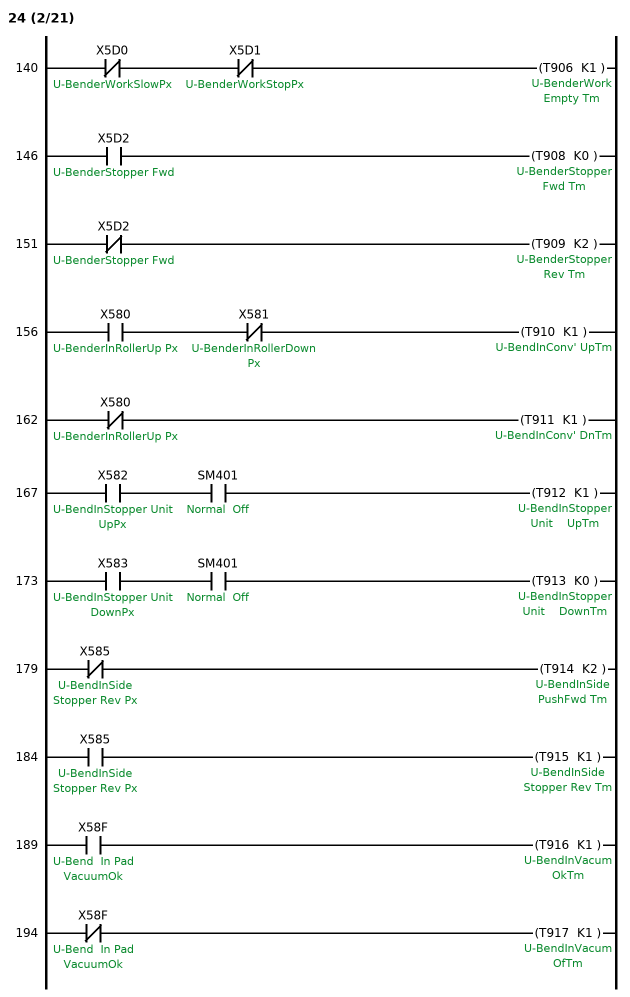
140   LDI     X5D0  ; U-BenderWorkSlowPx
      ANI     X5D1  ; U-BenderWorkStopPx
      OUT     T906 K1  ; U-BenderWork    Empty Tm
146   LD      X5D2  ; U-BenderStopper Fwd
      OUT     T908 K0  ; U-BenderStopper Fwd Tm
151   LDI     X5D2  ; U-BenderStopper Fwd
      OUT     T909 K2  ; U-BenderStopper Rev Tm
156   LD      X580  ; U-BenderInRollerUp Px
      ANI     X581  ; U-BenderInRollerDown Px
      OUT     T910 K1  ; U-BendInConv' UpTm
162   LDI     X580  ; U-BenderInRollerUp Px
      OUT     T911 K1  ; U-BendInConv' DnTm
167   LD      X582  ; U-BendInStopper Unit    UpPx
      AND     SM401  ; Normal  Off
      OUT     T912 K1  ; U-BendInStopper Unit    UpTm
173   LD      X583  ; U-BendInStopper Unit    DownPx
      AND     SM401  ; Normal  Off
      OUT     T913 K0  ; U-BendInStopper Unit    DownTm
179   LDI     X585  ; U-BendInSide    Stopper Rev Px
      OUT     T914 K2  ; U-BendInSide    PushFwd Tm
184   LD      X585  ; U-BendInSide    Stopper Rev Px
      OUT     T915 K1  ; U-BendInSide    Stopper Rev Tm
189   LD      X58F  ; U-Bend  In Pad  VacuumOk
      OUT     T916 K1  ; U-BendInVacum OkTm
194   LDI     X58F  ; U-Bend  In Pad  VacuumOk
      OUT     T917 K1  ; U-BendInVacum OfTm
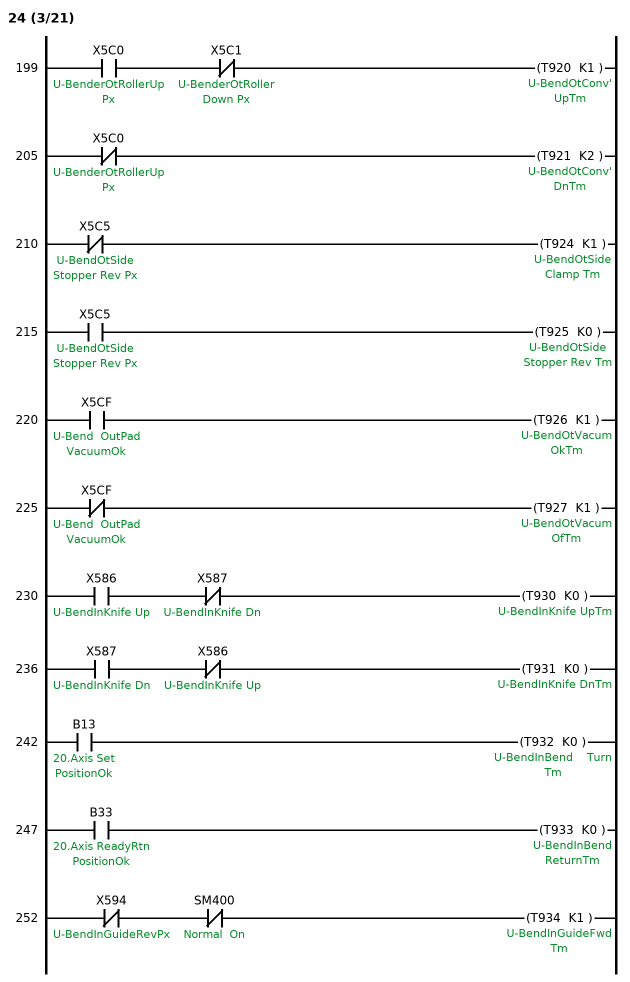
199   LD      X5C0  ; U-BenderOtRollerUp Px
      ANI     X5C1  ; U-BenderOtRollerDown Px
      OUT     T920 K1  ; U-BendOtConv' UpTm
205   LDI     X5C0  ; U-BenderOtRollerUp Px
      OUT     T921 K2  ; U-BendOtConv' DnTm
210   LDI     X5C5  ; U-BendOtSide    Stopper Rev Px
      OUT     T924 K1  ; U-BendOtSide    Clamp Tm
215   LD      X5C5  ; U-BendOtSide    Stopper Rev Px
      OUT     T925 K0  ; U-BendOtSide    Stopper Rev Tm
220   LD      X5CF  ; U-Bend  OutPad  VacuumOk
      OUT     T926 K1  ; U-BendOtVacum OkTm
225   LDI     X5CF  ; U-Bend  OutPad  VacuumOk
      OUT     T927 K1  ; U-BendOtVacum OfTm
230   LD      X586  ; U-BendInKnife Up
      ANI     X587  ; U-BendInKnife Dn
      OUT     T930 K0  ; U-BendInKnife UpTm
236   LD      X587  ; U-BendInKnife Dn
      ANI     X586  ; U-BendInKnife Up
      OUT     T931 K0  ; U-BendInKnife DnTm
242   LD      B13  ; 20.Axis Set     PositionOk
      OUT     T932 K0  ; U-BendInBend    Turn Tm
247   LD      B33  ; 20.Axis ReadyRtnPositionOk
      OUT     T933 K0  ; U-BendInBend    ReturnTm
252   LDI     X594  ; U-BendInGuideRevPx
      ANI     SM400  ; Normal  On
      OUT     T934 K1  ; U-BendInGuideFwdTm
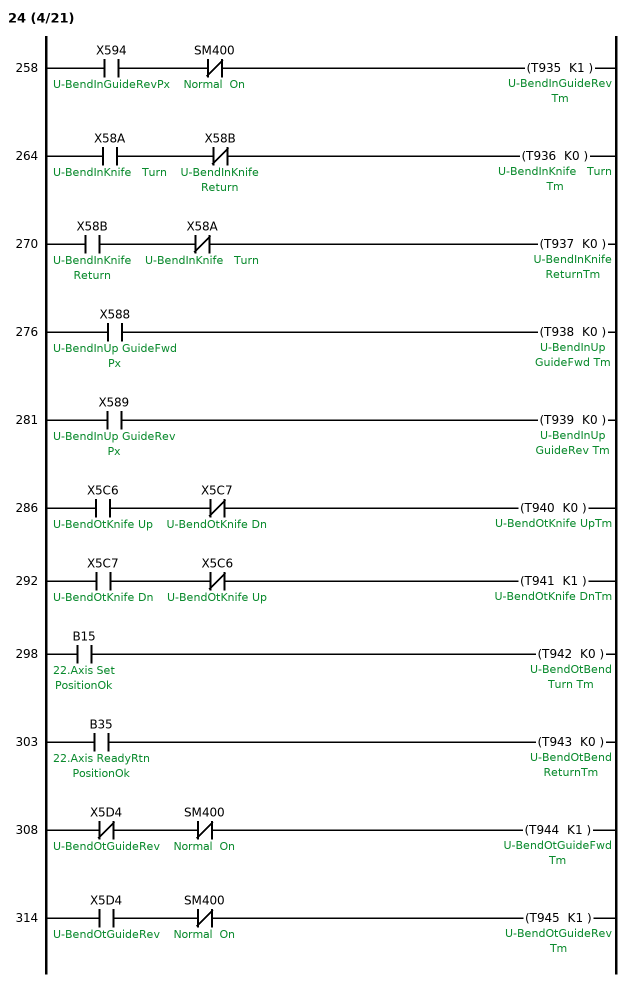
258   LD      X594  ; U-BendInGuideRevPx
      ANI     SM400  ; Normal  On
      OUT     T935 K1  ; U-BendInGuideRevTm
264   LD      X58A  ; U-BendInKnife   Turn
      ANI     X58B  ; U-BendInKnife   Return
      OUT     T936 K0  ; U-BendInKnife   Turn Tm
270   LD      X58B  ; U-BendInKnife   Return
      ANI     X58A  ; U-BendInKnife   Turn
      OUT     T937 K0  ; U-BendInKnife   ReturnTm
276   LD      X588  ; U-BendInUp GuideFwd Px
      OUT     T938 K0  ; U-BendInUp GuideFwd Tm
281   LD      X589  ; U-BendInUp GuideRev Px
      OUT     T939 K0  ; U-BendInUp GuideRev Tm
286   LD      X5C6  ; U-BendOtKnife Up
      ANI     X5C7  ; U-BendOtKnife Dn
      OUT     T940 K0  ; U-BendOtKnife UpTm
292   LD      X5C7  ; U-BendOtKnife Dn
      ANI     X5C6  ; U-BendOtKnife Up
      OUT     T941 K1  ; U-BendOtKnife DnTm
298   LD      B15  ; 22.Axis Set     PositionOk
      OUT     T942 K0  ; U-BendOtBend    Turn Tm
303   LD      B35  ; 22.Axis ReadyRtnPositionOk
      OUT     T943 K0  ; U-BendOtBend    ReturnTm
308   LDI     X5D4  ; U-BendOtGuideRev
      ANI     SM400  ; Normal  On
      OUT     T944 K1  ; U-BendOtGuideFwdTm
314   LD      X5D4  ; U-BendOtGuideRev
      ANI     SM400  ; Normal  On
      OUT     T945 K1  ; U-BendOtGuideRevTm
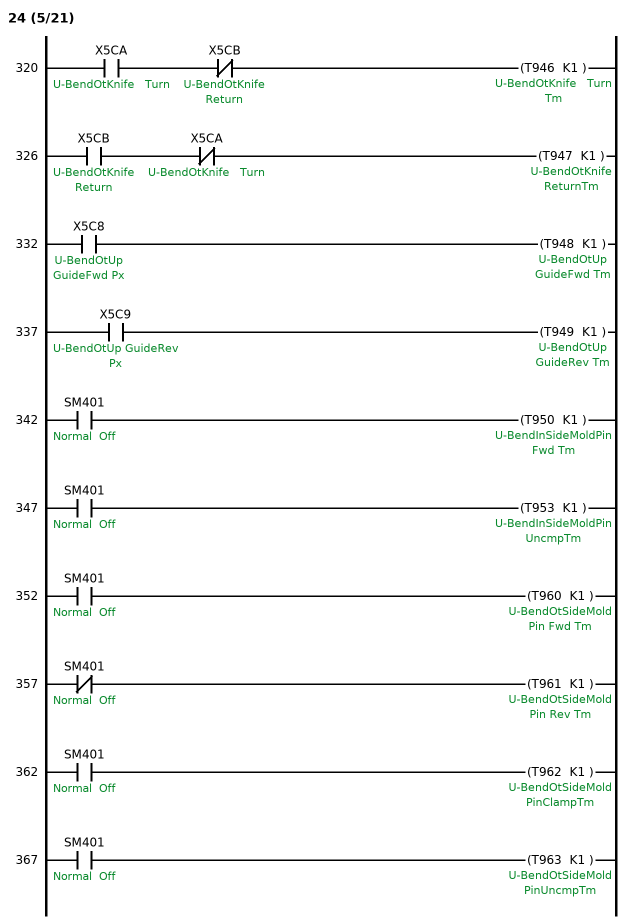
320   LD      X5CA  ; U-BendOtKnife   Turn
      ANI     X5CB  ; U-BendOtKnife   Return
      OUT     T946 K1  ; U-BendOtKnife   Turn Tm
326   LD      X5CB  ; U-BendOtKnife   Return
      ANI     X5CA  ; U-BendOtKnife   Turn
      OUT     T947 K1  ; U-BendOtKnife   ReturnTm
332   LD      X5C8  ; U-BendOtUp GuideFwd Px
      OUT     T948 K1  ; U-BendOtUp GuideFwd Tm
337   LD      X5C9  ; U-BendOtUp GuideRev Px
      OUT     T949 K1  ; U-BendOtUp GuideRev Tm
342   LD      SM401  ; Normal  Off
      OUT     T950 K1  ; U-BendInSideMoldPin Fwd Tm
347   LD      SM401  ; Normal  Off
      OUT     T953 K1  ; U-BendInSideMoldPinUncmpTm
352   LD      SM401  ; Normal  Off
      OUT     T960 K1  ; U-BendOtSideMoldPin Fwd Tm
357   LDI     SM401  ; Normal  Off
      OUT     T961 K1  ; U-BendOtSideMoldPin Rev Tm
362   LD      SM401  ; Normal  Off
      OUT     T962 K1  ; U-BendOtSideMoldPinClampTm
367   LD      SM401  ; Normal  Off
      OUT     T963 K1  ; U-BendOtSideMoldPinUncmpTm
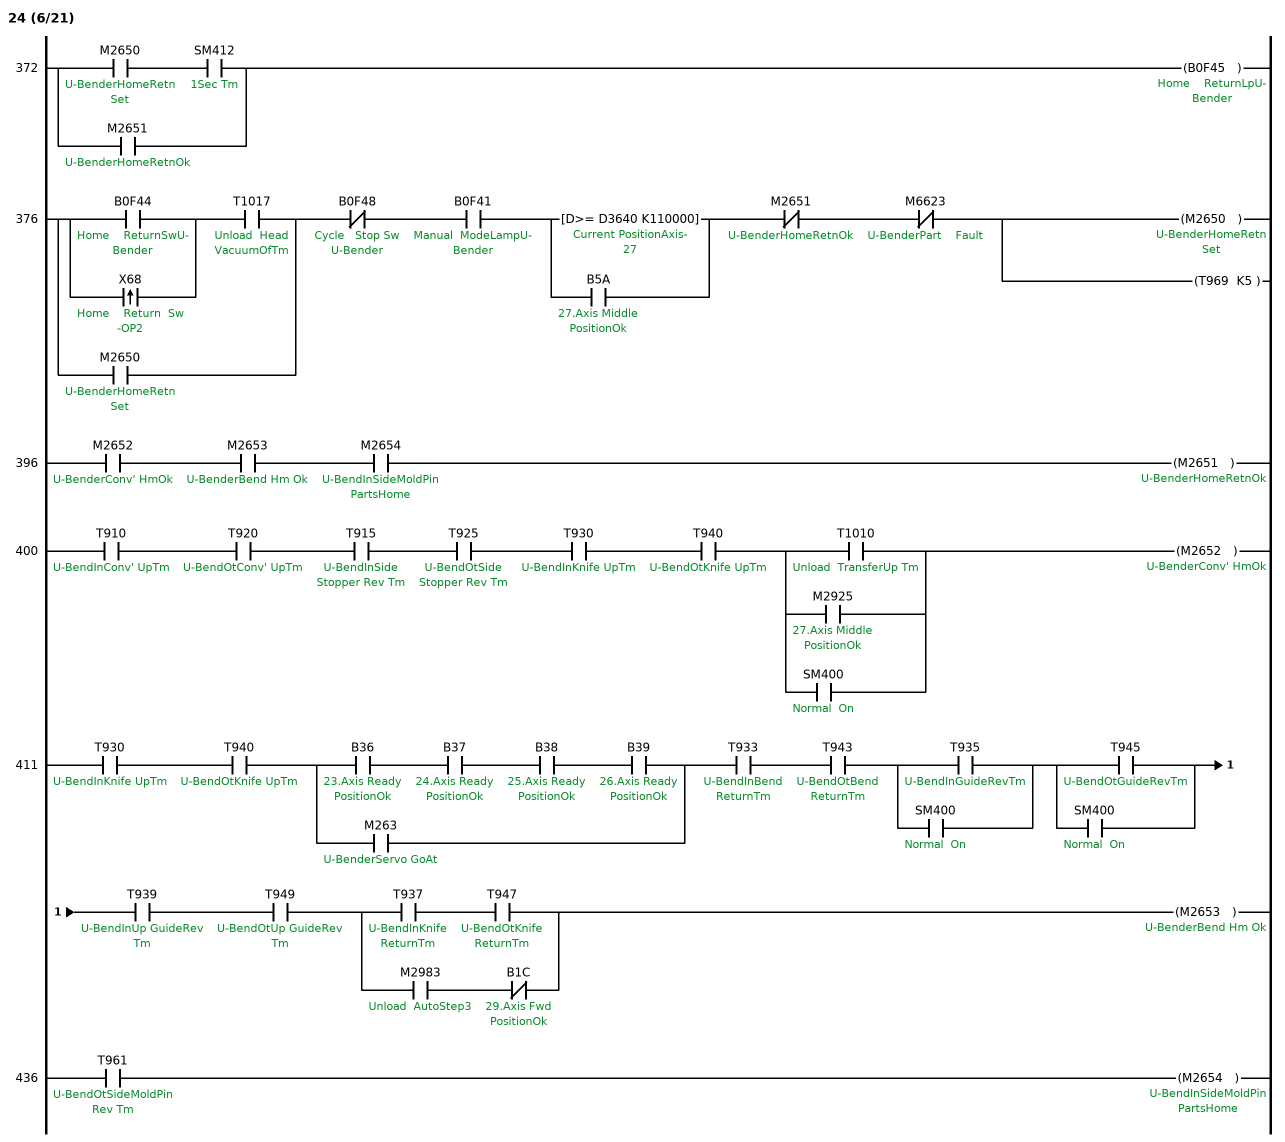
372   LD      M2650  ; U-BenderHomeRetnSet
      AND     SM412  ; 1Sec Tm
      OR      M2651  ; U-BenderHomeRetnOk
      OUT     B0F45  ; Home    ReturnLpU-Bender
376   LD      B0F44  ; Home    ReturnSwU-Bender
      ORP     X68  ; Home    Return  Sw -OP2
      AND     T1017  ; Unload  Head    VacuumOfTm
      OR      M2650  ; U-BenderHomeRetnSet
      ANI     B0F48  ; Cycle   Stop Sw U-Bender
      AND     B0F41  ; Manual  ModeLampU-Bender
      LDD>=   D3640 K110000  ; Current PositionAxis-27
      OR      B5A  ; 27.Axis Middle  PositionOk
      ANB
      ANI     M2651  ; U-BenderHomeRetnOk
      ANI     M6623  ; U-BenderPart    Fault
      OUT     M2650  ; U-BenderHomeRetnSet
      OUT     T969 K5
396   LD      M2652  ; U-BenderConv' HmOk
      AND     M2653  ; U-BenderBend Hm Ok
      AND     M2654  ; U-BendInSideMoldPinPartsHome
      OUT     M2651  ; U-BenderHomeRetnOk
400   LD      T910  ; U-BendInConv' UpTm
      AND     T920  ; U-BendOtConv' UpTm
      AND     T915  ; U-BendInSide    Stopper Rev Tm
      AND     T925  ; U-BendOtSide    Stopper Rev Tm
      AND     T930  ; U-BendInKnife UpTm
      AND     T940  ; U-BendOtKnife UpTm
      LD      T1010  ; Unload  TransferUp Tm
      OR      M2925  ; 27.Axis Middle  PositionOk
      OR      SM400  ; Normal  On
      ANB
      OUT     M2652  ; U-BenderConv' HmOk
411   LD      T930  ; U-BendInKnife UpTm
      AND     T940  ; U-BendOtKnife UpTm
      LD      B36  ; 23.Axis Ready   PositionOk
      AND     B37  ; 24.Axis Ready   PositionOk
      AND     B38  ; 25.Axis Ready   PositionOk
      AND     B39  ; 26.Axis Ready   PositionOk
      OR      M263  ; U-BenderServo GoAt
      ANB
      AND     T933  ; U-BendInBend    ReturnTm
      AND     T943  ; U-BendOtBend    ReturnTm
      LD      T935  ; U-BendInGuideRevTm
      OR      SM400  ; Normal  On
      ANB
      LD      T945  ; U-BendOtGuideRevTm
      OR      SM400  ; Normal  On
      ANB
      AND     T939  ; U-BendInUp GuideRev Tm
      AND     T949  ; U-BendOtUp GuideRev Tm
      LD      T937  ; U-BendInKnife   ReturnTm
      AND     T947  ; U-BendOtKnife   ReturnTm
      LD      M2983  ; Unload  AutoStep3
      ANI     B1C  ; 29.Axis Fwd     PositionOk
      ORB
      ANB
      OUT     M2653  ; U-BenderBend Hm Ok
436   LD      T961  ; U-BendOtSideMoldPin Rev Tm
      OUT     M2654  ; U-BendInSideMoldPinPartsHome
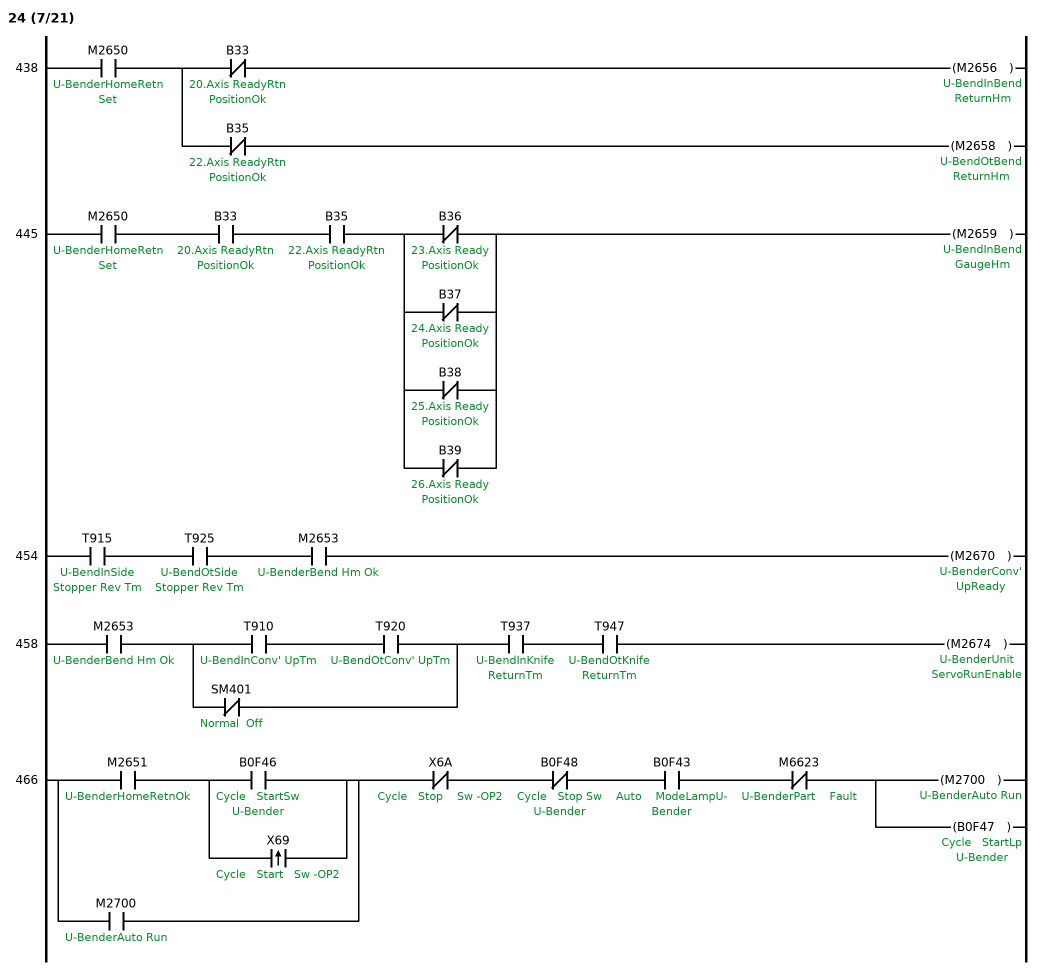
438   LD      M2650  ; U-BenderHomeRetnSet
      MPS
      ANI     B33  ; 20.Axis ReadyRtnPositionOk
      OUT     M2656  ; U-BendInBend    ReturnHm
      MPP
      ANI     B35  ; 22.Axis ReadyRtnPositionOk
      OUT     M2658  ; U-BendOtBend    ReturnHm
445   LD      M2650  ; U-BenderHomeRetnSet
      AND     B33  ; 20.Axis ReadyRtnPositionOk
      AND     B35  ; 22.Axis ReadyRtnPositionOk
      LDI     B36  ; 23.Axis Ready   PositionOk
      ORI     B37  ; 24.Axis Ready   PositionOk
      ORI     B38  ; 25.Axis Ready   PositionOk
      ORI     B39  ; 26.Axis Ready   PositionOk
      ANB
      OUT     M2659  ; U-BendInBend    GaugeHm
454   LD      T915  ; U-BendInSide    Stopper Rev Tm
      AND     T925  ; U-BendOtSide    Stopper Rev Tm
      AND     M2653  ; U-BenderBend Hm Ok
      OUT     M2670  ; U-BenderConv' UpReady
458   LD      M2653  ; U-BenderBend Hm Ok
      LD      T910  ; U-BendInConv' UpTm
      AND     T920  ; U-BendOtConv' UpTm
      ORI     SM401  ; Normal  Off
      ANB
      AND     T937  ; U-BendInKnife   ReturnTm
      AND     T947  ; U-BendOtKnife   ReturnTm
      OUT     M2674  ; U-BenderUnit    ServoRunEnable
466   LD      M2651  ; U-BenderHomeRetnOk
      LD      B0F46  ; Cycle   StartSw U-Bender
      ORP     X69  ; Cycle   Start   Sw -OP2
      ANB
      OR      M2700  ; U-BenderAuto Run
      ANI     X6A  ; Cycle   Stop    Sw -OP2
      ANI     B0F48  ; Cycle   Stop Sw U-Bender
      AND     B0F43  ; Auto    ModeLampU-Bender
      ANI     M6623  ; U-BenderPart    Fault
      OUT     M2700  ; U-BenderAuto Run
      OUT     B0F47  ; Cycle   StartLp U-Bender
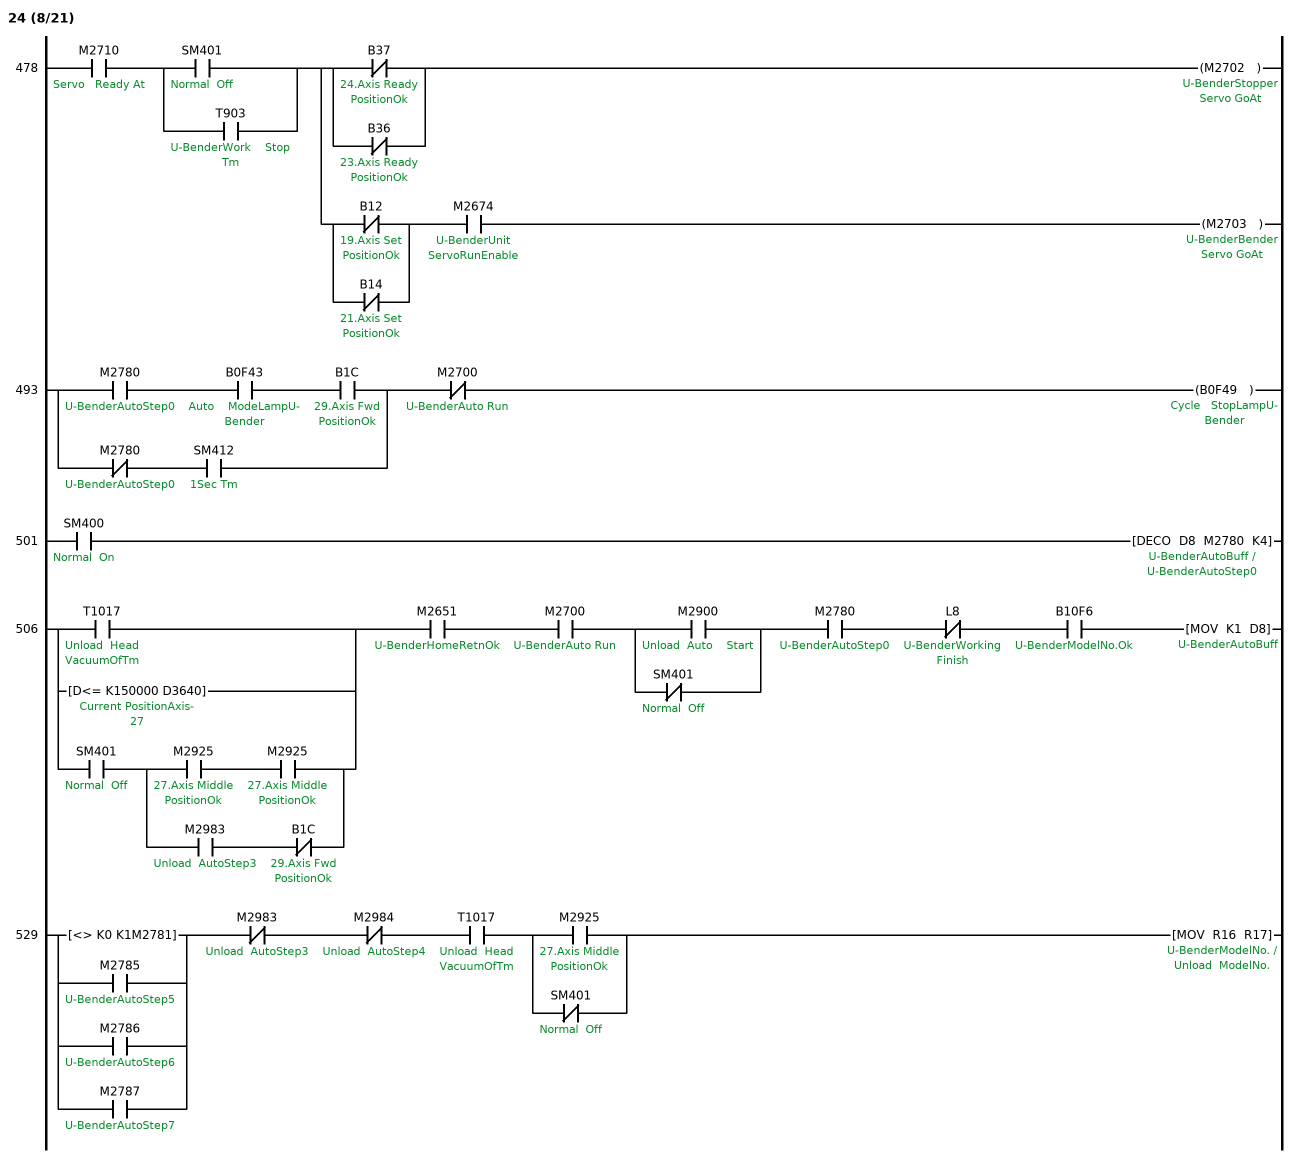
478   LD      M2710  ; Servo   Ready At
      LD      SM401  ; Normal  Off
      OR      T903  ; U-BenderWork    Stop Tm
      ANB
      MPS
      LDI     B37  ; 24.Axis Ready   PositionOk
      ORI     B36  ; 23.Axis Ready   PositionOk
      ANB
      OUT     M2702  ; U-BenderStopper Servo GoAt
      MPP
      LDI     B12  ; 19.Axis Set     PositionOk
      ORI     B14  ; 21.Axis Set     PositionOk
      ANB
      AND     M2674  ; U-BenderUnit    ServoRunEnable
      OUT     M2703  ; U-BenderBender  Servo GoAt
493   LD      M2780  ; U-BenderAutoStep0
      AND     B0F43  ; Auto    ModeLampU-Bender
      AND     B1C  ; 29.Axis Fwd     PositionOk
      LDI     M2780  ; U-BenderAutoStep0
      AND     SM412  ; 1Sec Tm
      ORB
      ANI     M2700  ; U-BenderAuto Run
      OUT     B0F49  ; Cycle   StopLampU-Bender
501   LD      SM400  ; Normal  On
      DECO    D8 M2780 K4  ; U-BenderAutoBuff
506   LD      T1017  ; Unload  Head    VacuumOfTm
      ORD<=   K150000 D3640  ; Current PositionAxis-27
      LD      SM401  ; Normal  Off
      LD      M2925  ; 27.Axis Middle  PositionOk
      AND     M2925  ; 27.Axis Middle  PositionOk
      LD      M2983  ; Unload  AutoStep3
      ANI     B1C  ; 29.Axis Fwd     PositionOk
      ORB
      ANB
      ORB
      AND     M2651  ; U-BenderHomeRetnOk
      AND     M2700  ; U-BenderAuto Run
      LD      M2900  ; Unload  Auto    Start
      ORI     SM401  ; Normal  Off
      ANB
      AND     M2780  ; U-BenderAutoStep0
      ANI     L8  ; U-BenderWorking Finish
      AND     B10F6  ; U-BenderModelNo.Ok
      MOV     K1 D8
529   LD<>    K0 K1M2781  ; U-BenderAutoStep1
      OR      M2785  ; U-BenderAutoStep5
      OR      M2786  ; U-BenderAutoStep6
      OR      M2787  ; U-BenderAutoStep7
      ANI     M2983  ; Unload  AutoStep3
      ANI     M2984  ; Unload  AutoStep4
      AND     T1017  ; Unload  Head    VacuumOfTm
      LD      M2925  ; 27.Axis Middle  PositionOk
      ORI     SM401  ; Normal  Off
      ANB
      MOV     R16 R17  ; U-BenderModelNo. / Unload  ModelNo.
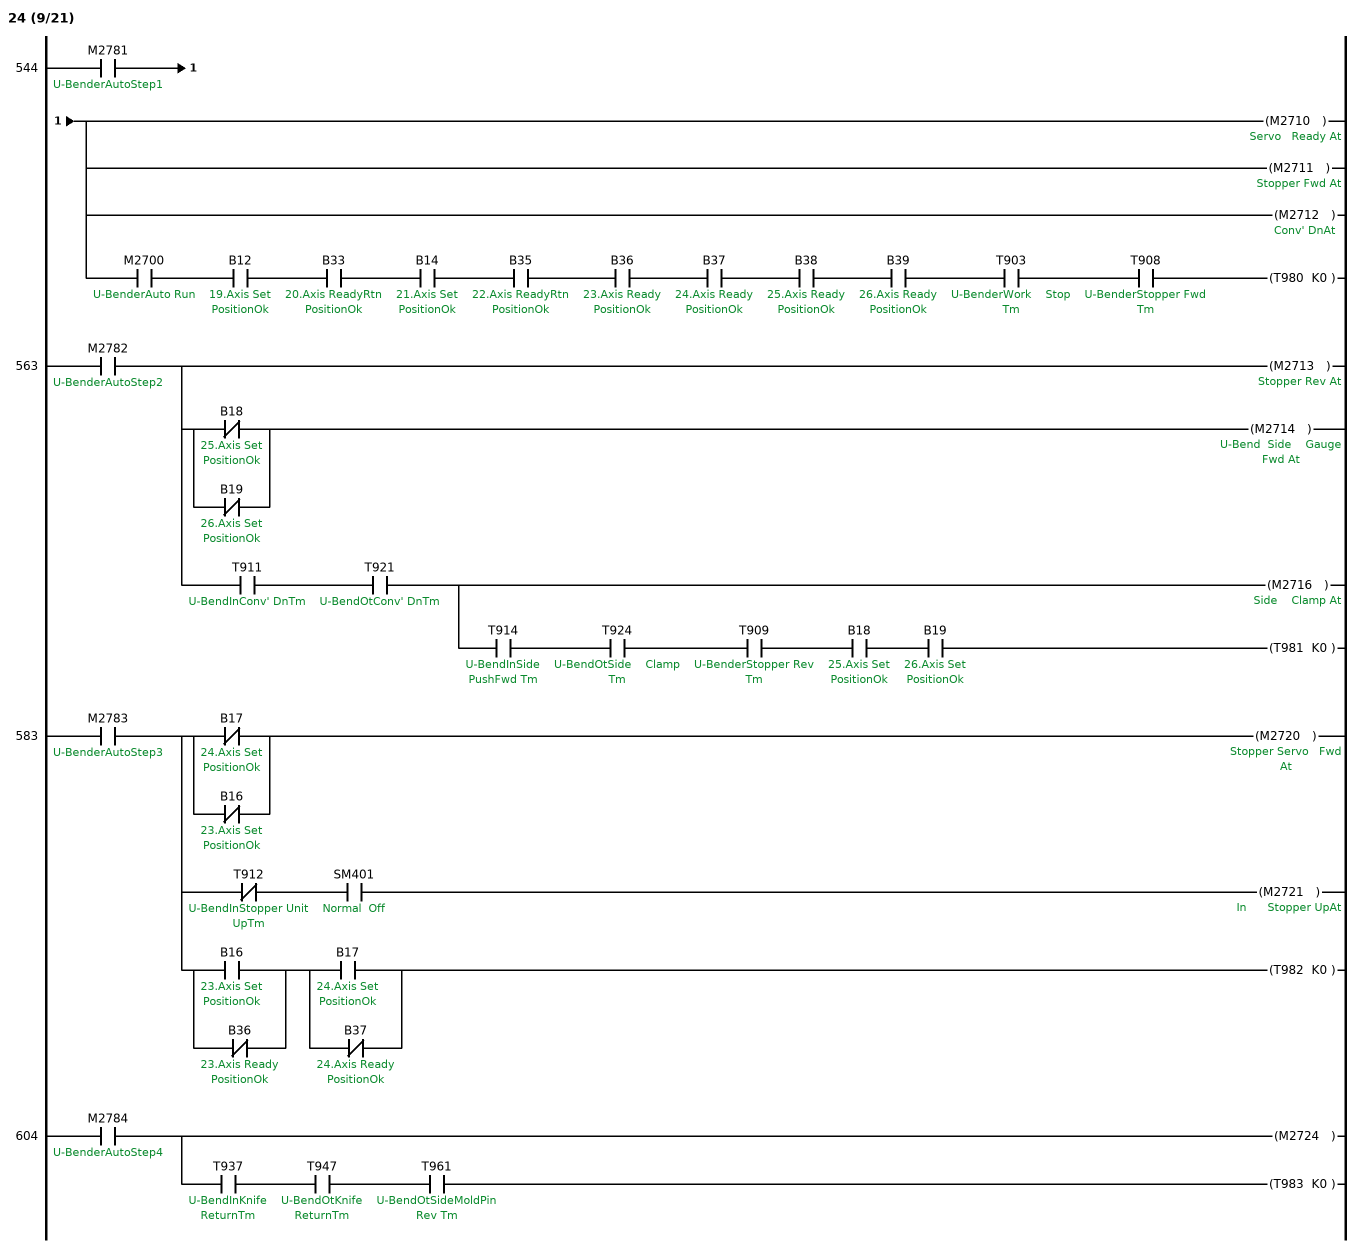
544   LD      M2781  ; U-BenderAutoStep1
      OUT     M2710  ; Servo   Ready At
      OUT     M2711  ; Stopper Fwd At
      OUT     M2712  ; Conv' DnAt
      AND     M2700  ; U-BenderAuto Run
      AND     B12  ; 19.Axis Set     PositionOk
      AND     B33  ; 20.Axis ReadyRtnPositionOk
      AND     B14  ; 21.Axis Set     PositionOk
      AND     B35  ; 22.Axis ReadyRtnPositionOk
      AND     B36  ; 23.Axis Ready   PositionOk
      AND     B37  ; 24.Axis Ready   PositionOk
      AND     B38  ; 25.Axis Ready   PositionOk
      AND     B39  ; 26.Axis Ready   PositionOk
      AND     T903  ; U-BenderWork    Stop Tm
      AND     T908  ; U-BenderStopper Fwd Tm
      OUT     T980 K0
563   LD      M2782  ; U-BenderAutoStep2
      OUT     M2713  ; Stopper Rev At
      MPS
      LDI     B18  ; 25.Axis Set     PositionOk
      ORI     B19  ; 26.Axis Set     PositionOk
      ANB
      OUT     M2714  ; U-Bend  Side    Gauge   Fwd At
      MPP
      AND     T911  ; U-BendInConv' DnTm
      AND     T921  ; U-BendOtConv' DnTm
      OUT     M2716  ; Side    Clamp At
      AND     T914  ; U-BendInSide    PushFwd Tm
      AND     T924  ; U-BendOtSide    Clamp Tm
      AND     T909  ; U-BenderStopper Rev Tm
      AND     B18  ; 25.Axis Set     PositionOk
      AND     B19  ; 26.Axis Set     PositionOk
      OUT     T981 K0
583   LD      M2783  ; U-BenderAutoStep3
      MPS
      LDI     B17  ; 24.Axis Set     PositionOk
      ORI     B16  ; 23.Axis Set     PositionOk
      ANB
      OUT     M2720  ; Stopper Servo   Fwd At
      MRD
      ANI     T912  ; U-BendInStopper Unit    UpTm
      AND     SM401  ; Normal  Off
      OUT     M2721  ; In      Stopper UpAt
      MPP
      LD      B16  ; 23.Axis Set     PositionOk
      ORI     B36  ; 23.Axis Ready   PositionOk
      ANB
      LD      B17  ; 24.Axis Set     PositionOk
      ORI     B37  ; 24.Axis Ready   PositionOk
      ANB
      OUT     T982 K0
604   LD      M2784  ; U-BenderAutoStep4
      OUT     M2724
      AND     T937  ; U-BendInKnife   ReturnTm
      AND     T947  ; U-BendOtKnife   ReturnTm
      AND     T961  ; U-BendOtSideMoldPin Rev Tm
      OUT     T983 K0
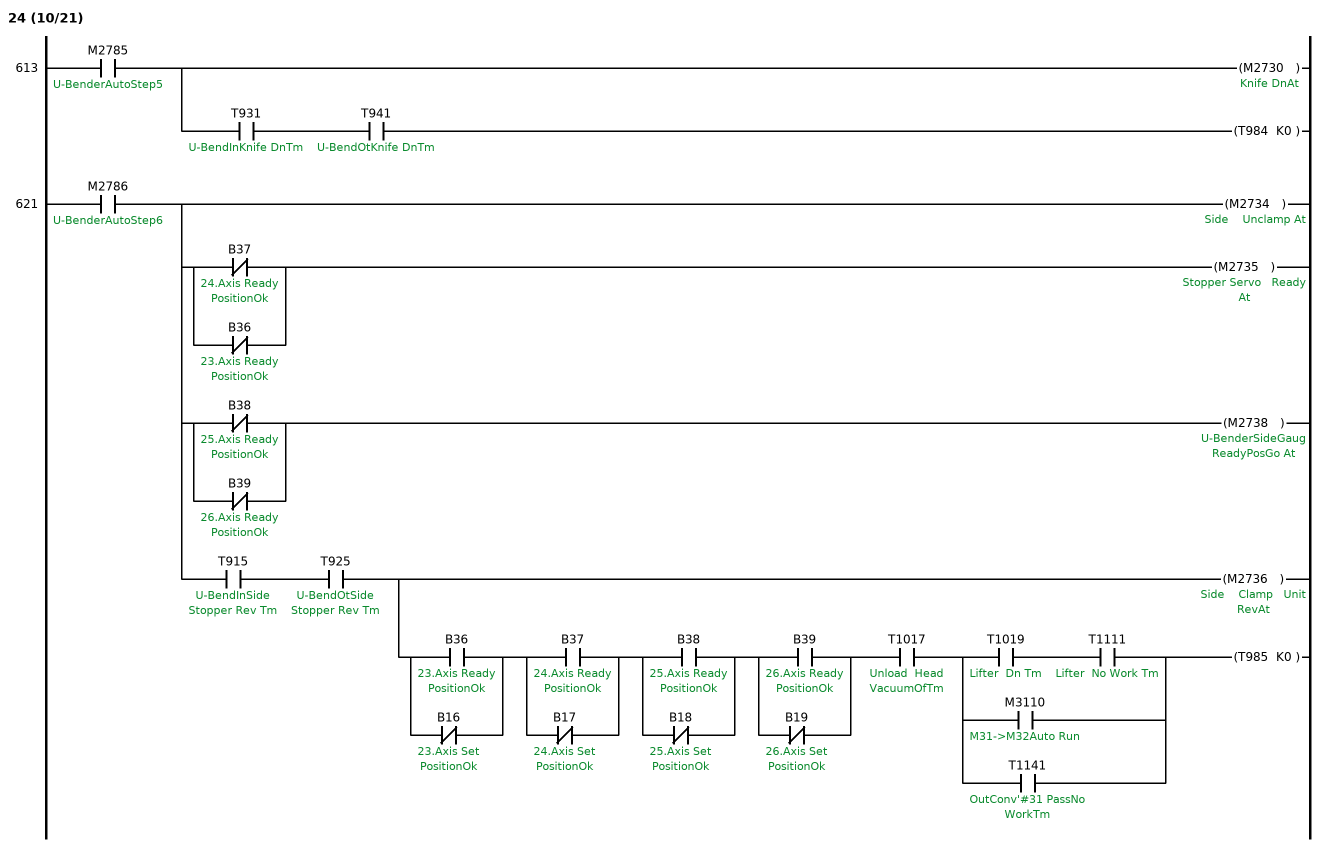
613   LD      M2785  ; U-BenderAutoStep5
      OUT     M2730  ; Knife DnAt
      AND     T931  ; U-BendInKnife DnTm
      AND     T941  ; U-BendOtKnife DnTm
      OUT     T984 K0
621   LD      M2786  ; U-BenderAutoStep6
      OUT     M2734  ; Side    Unclamp At
      MPS
      LDI     B37  ; 24.Axis Ready   PositionOk
      ORI     B36  ; 23.Axis Ready   PositionOk
      ANB
      OUT     M2735  ; Stopper Servo   Ready At
      MRD
      LDI     B38  ; 25.Axis Ready   PositionOk
      ORI     B39  ; 26.Axis Ready   PositionOk
      ANB
      OUT     M2738  ; U-BenderSideGaugReadyPosGo At
      MPP
      AND     T915  ; U-BendInSide    Stopper Rev Tm
      AND     T925  ; U-BendOtSide    Stopper Rev Tm
      OUT     M2736  ; Side    Clamp   Unit RevAt
      LD      B36  ; 23.Axis Ready   PositionOk
      ORI     B16  ; 23.Axis Set     PositionOk
      ANB
      LD      B37  ; 24.Axis Ready   PositionOk
      ORI     B17  ; 24.Axis Set     PositionOk
      ANB
      LD      B38  ; 25.Axis Ready   PositionOk
      ORI     B18  ; 25.Axis Set     PositionOk
      ANB
      LD      B39  ; 26.Axis Ready   PositionOk
      ORI     B19  ; 26.Axis Set     PositionOk
      ANB
      AND     T1017  ; Unload  Head    VacuumOfTm
      LD      T1019  ; Lifter  Dn Tm
      AND     T1111  ; Lifter  No Work Tm
      OR      M3110  ; M31->M32Auto Run
      OR      T1141  ; OutConv'#31 PassNo  WorkTm
      ANB
      OUT     T985 K0
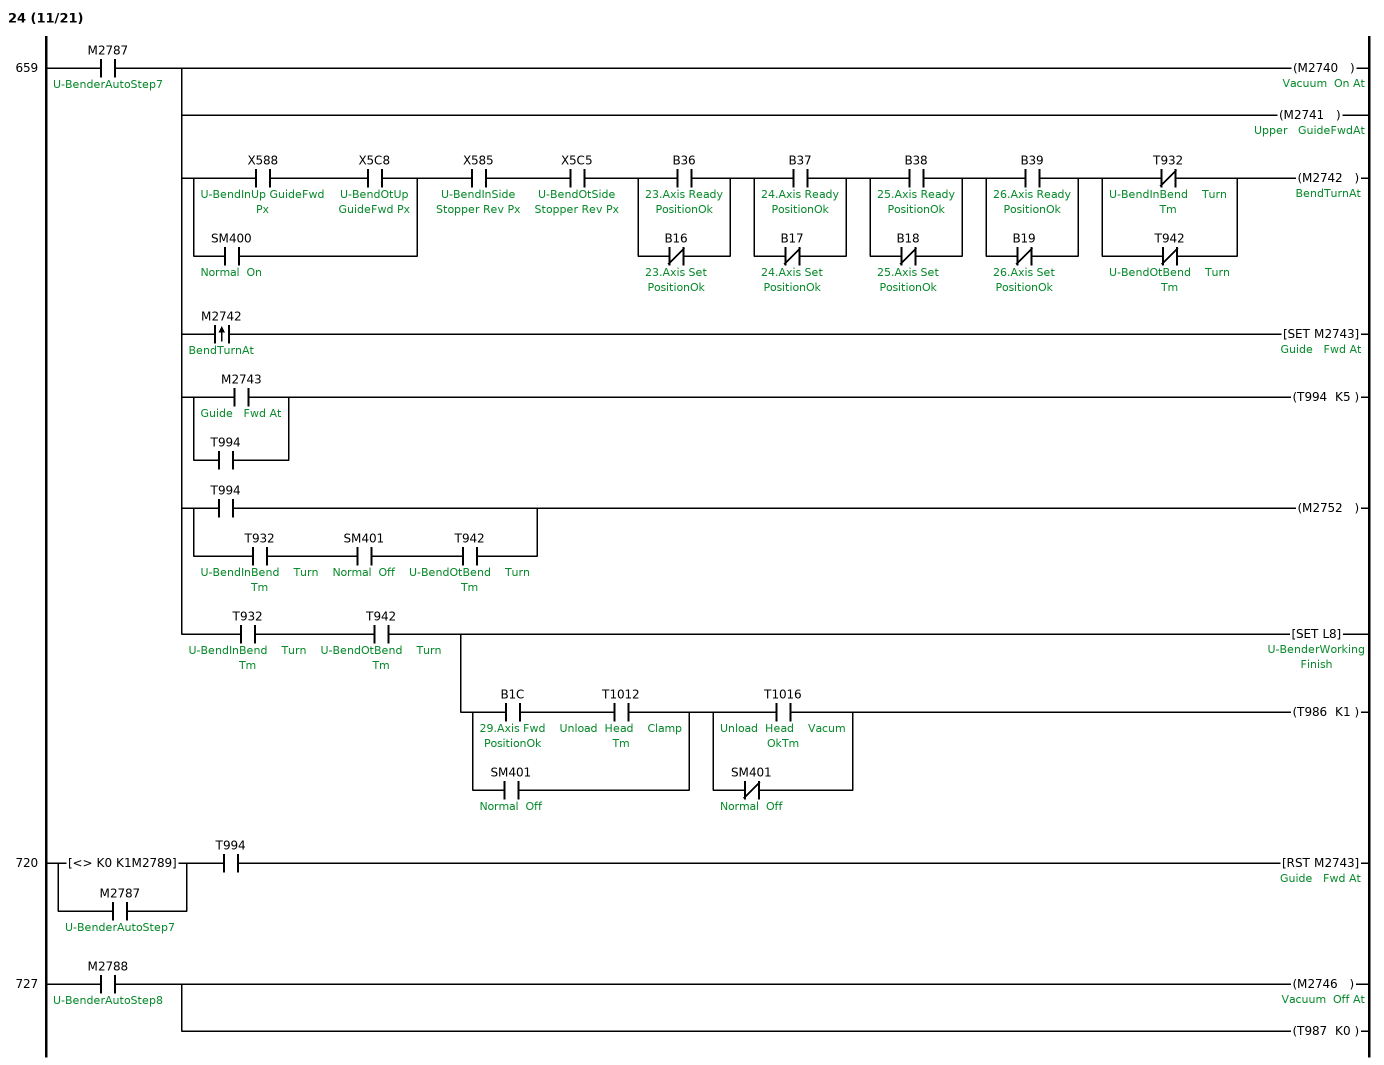
659   LD      M2787  ; U-BenderAutoStep7
      OUT     M2740  ; Vacuum  On At
      OUT     M2741  ; Upper   GuideFwdAt
      MPS
      LD      X588  ; U-BendInUp GuideFwd Px
      AND     X5C8  ; U-BendOtUp GuideFwd Px
      OR      SM400  ; Normal  On
      ANB
      AND     X585  ; U-BendInSide    Stopper Rev Px
      AND     X5C5  ; U-BendOtSide    Stopper Rev Px
      LD      B36  ; 23.Axis Ready   PositionOk
      ORI     B16  ; 23.Axis Set     PositionOk
      ANB
      LD      B37  ; 24.Axis Ready   PositionOk
      ORI     B17  ; 24.Axis Set     PositionOk
      ANB
      LD      B38  ; 25.Axis Ready   PositionOk
      ORI     B18  ; 25.Axis Set     PositionOk
      ANB
      LD      B39  ; 26.Axis Ready   PositionOk
      ORI     B19  ; 26.Axis Set     PositionOk
      ANB
      LDI     T932  ; U-BendInBend    Turn Tm
      ORI     T942  ; U-BendOtBend    Turn Tm
      ANB
      OUT     M2742  ; BendTurnAt
      MRD
      ANDP    M2742  ; BendTurnAt
      SET     M2743  ; Guide   Fwd At
      MRD
      LD      M2743  ; Guide   Fwd At
      OR      T994
      ANB
      OUT     T994 K5
      MRD
      LD      T994
      LD      T932  ; U-BendInBend    Turn Tm
      AND     SM401  ; Normal  Off
      AND     T942  ; U-BendOtBend    Turn Tm
      ORB
      ANB
      OUT     M2752
      MPP
      AND     T932  ; U-BendInBend    Turn Tm
      AND     T942  ; U-BendOtBend    Turn Tm
      SET     L8  ; U-BenderWorking Finish
      LD      B1C  ; 29.Axis Fwd     PositionOk
      AND     T1012  ; Unload  Head    Clamp Tm
      OR      SM401  ; Normal  Off
      ANB
      LD      T1016  ; Unload  Head    Vacum OkTm
      ORI     SM401  ; Normal  Off
      ANB
      OUT     T986 K1
720   LD<>    K0 K1M2789  ; U-BenderAutoStep9
      OR      M2787  ; U-BenderAutoStep7
      AND     T994
      RST     M2743  ; Guide   Fwd At
727   LD      M2788  ; U-BenderAutoStep8
      OUT     M2746  ; Vacuum  Off At
      OUT     T987 K0
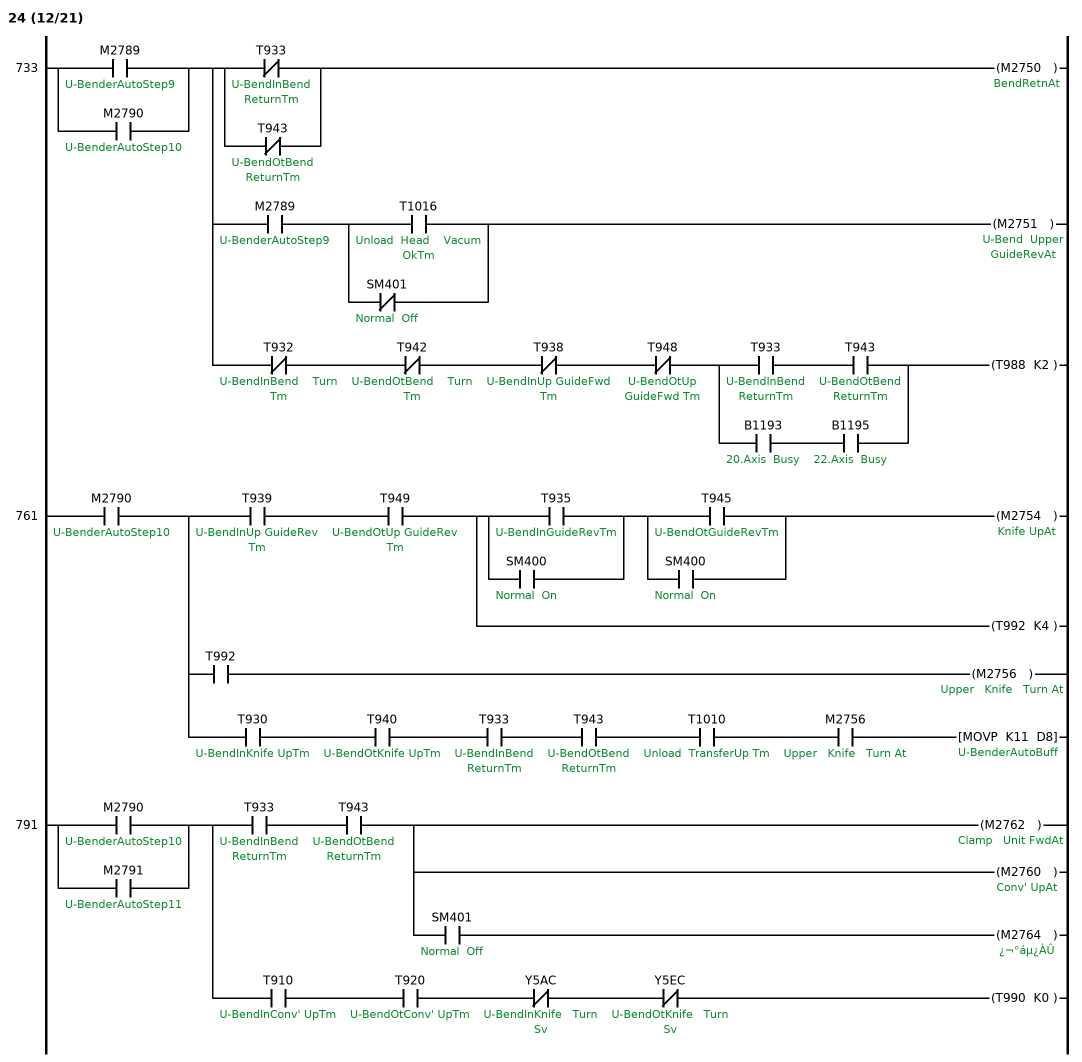
733   LD      M2789  ; U-BenderAutoStep9
      OR      M2790  ; U-BenderAutoStep10
      MPS
      LDI     T933  ; U-BendInBend    ReturnTm
      ORI     T943  ; U-BendOtBend    ReturnTm
      ANB
      OUT     M2750  ; BendRetnAt
      MRD
      AND     M2789  ; U-BenderAutoStep9
      LD      T1016  ; Unload  Head    Vacum OkTm
      ORI     SM401  ; Normal  Off
      ANB
      OUT     M2751  ; U-Bend  Upper   GuideRevAt
      MPP
      ANI     T932  ; U-BendInBend    Turn Tm
      ANI     T942  ; U-BendOtBend    Turn Tm
      ANI     T938  ; U-BendInUp GuideFwd Tm
      ANI     T948  ; U-BendOtUp GuideFwd Tm
      LD      T933  ; U-BendInBend    ReturnTm
      AND     T943  ; U-BendOtBend    ReturnTm
      LD      B1193  ; 20.Axis  Busy
      AND     B1195  ; 22.Axis  Busy
      ORB
      ANB
      OUT     T988 K2
761   LD      M2790  ; U-BenderAutoStep10
      MPS
      AND     T939  ; U-BendInUp GuideRev Tm
      AND     T949  ; U-BendOtUp GuideRev Tm
      MPS
      LD      T935  ; U-BendInGuideRevTm
      OR      SM400  ; Normal  On
      ANB
      LD      T945  ; U-BendOtGuideRevTm
      OR      SM400  ; Normal  On
      ANB
      OUT     M2754  ; Knife UpAt
      MPP
      OUT     T992 K4
      MRD
      AND     T992
      OUT     M2756  ; Upper   Knife   Turn At
      MPP
      AND     T930  ; U-BendInKnife UpTm
      AND     T940  ; U-BendOtKnife UpTm
      AND     T933  ; U-BendInBend    ReturnTm
      AND     T943  ; U-BendOtBend    ReturnTm
      AND     T1010  ; Unload  TransferUp Tm
      AND     M2756  ; Upper   Knife   Turn At
      MOVP    K11 D8
791   LD      M2790  ; U-BenderAutoStep10
      OR      M2791  ; U-BenderAutoStep11
      MPS
      AND     T933  ; U-BendInBend    ReturnTm
      AND     T943  ; U-BendOtBend    ReturnTm
      OUT     M2762  ; Clamp   Unit FwdAt
      OUT     M2760  ; Conv' UpAt
      AND     SM401  ; Normal  Off
      OUT     M2764  ; ¿¬°áµ¿ÀÛ
      MPP
      AND     T910  ; U-BendInConv' UpTm
      AND     T920  ; U-BendOtConv' UpTm
      ANI     Y5AC  ; U-BendInKnife   Turn Sv
      ANI     Y5EC  ; U-BendOtKnife   Turn Sv
      OUT     T990 K0
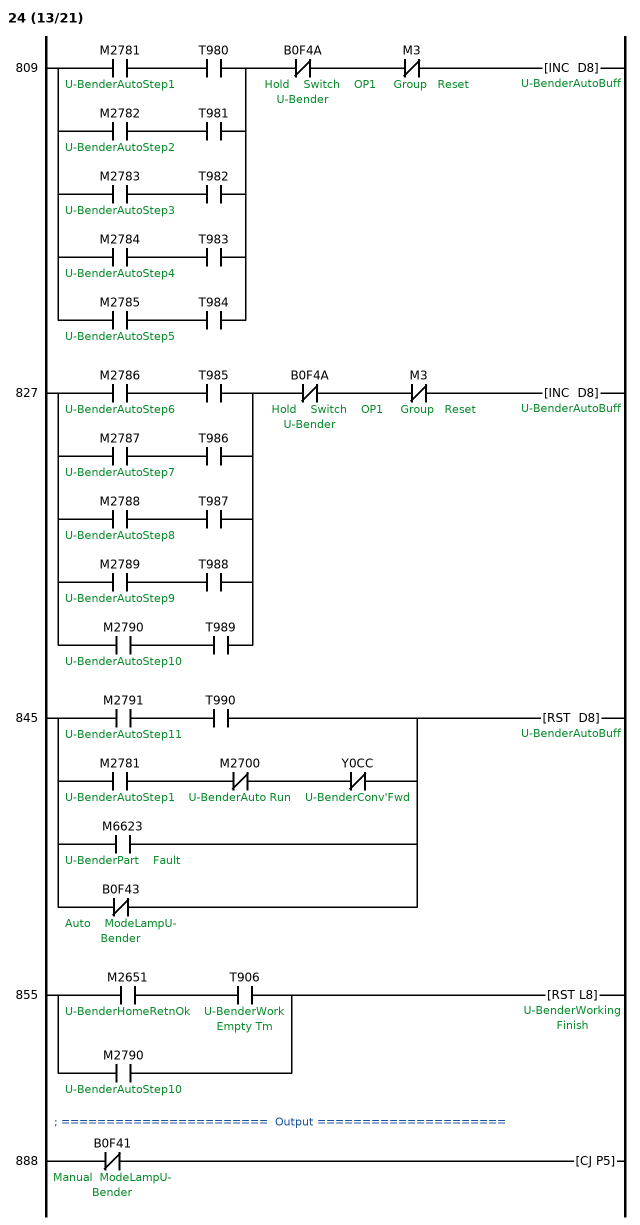
809   LD      M2781  ; U-BenderAutoStep1
      AND     T980
      LD      M2782  ; U-BenderAutoStep2
      AND     T981
      ORB
      LD      M2783  ; U-BenderAutoStep3
      AND     T982
      ORB
      LD      M2784  ; U-BenderAutoStep4
      AND     T983
      ORB
      LD      M2785  ; U-BenderAutoStep5
      AND     T984
      ORB
      ANI     B0F4A  ; Hold    Switch  U-Bender
      ANI     M3  ; OP1     Group   Reset
      INC     D8
827   LD      M2786  ; U-BenderAutoStep6
      AND     T985
      LD      M2787  ; U-BenderAutoStep7
      AND     T986
      ORB
      LD      M2788  ; U-BenderAutoStep8
      AND     T987
      ORB
      LD      M2789  ; U-BenderAutoStep9
      AND     T988
      ORB
      LD      M2790  ; U-BenderAutoStep10
      AND     T989
      ORB
      ANI     B0F4A  ; Hold    Switch  U-Bender
      ANI     M3  ; OP1     Group   Reset
      INC     D8
845   LD      M2791  ; U-BenderAutoStep11
      AND     T990
      LD      M2781  ; U-BenderAutoStep1
      ANI     M2700  ; U-BenderAuto Run
      ANI     Y0CC  ; U-BenderConv'Fwd
      ORB
      OR      M6623  ; U-BenderPart    Fault
      ORI     B0F43  ; Auto    ModeLampU-Bender
      RST     D8  ; U-BenderAutoBuff
855   LD      M2651  ; U-BenderHomeRetnOk
      AND     T906  ; U-BenderWork    Empty Tm
      OR      M2790  ; U-BenderAutoStep10
      RST     L8  ; U-BenderWorking Finish
; =======================  Output =====================
888   LDI     B0F41  ; Manual  ModeLampU-Bender
      CJ      P5
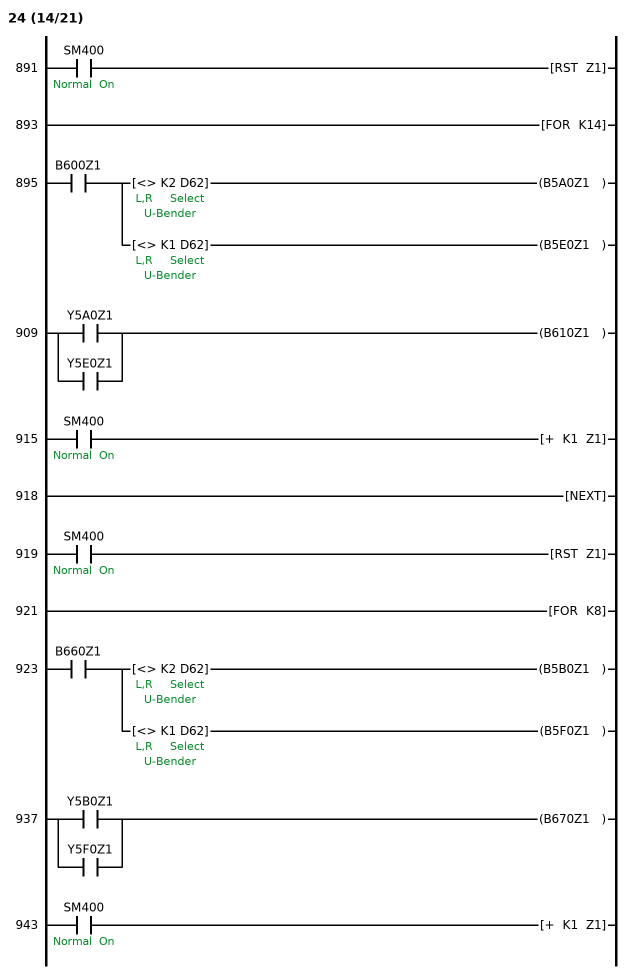
891   LD      SM400  ; Normal  On
      RST     Z1
893   FOR     K14
895   LD      B600Z1
      MPS
      AND<>   K2 D62  ; L,R     Select  U-Bender
      OUT     B5A0Z1
      MPP
      AND<>   K1 D62  ; L,R     Select  U-Bender
      OUT     B5E0Z1
909   LD      Y5A0Z1
      OR      Y5E0Z1
      OUT     B610Z1
915   LD      SM400  ; Normal  On
      +       K1 Z1
918   NEXT
919   LD      SM400  ; Normal  On
      RST     Z1
921   FOR     K8
923   LD      B660Z1
      MPS
      AND<>   K2 D62  ; L,R     Select  U-Bender
      OUT     B5B0Z1
      MPP
      AND<>   K1 D62  ; L,R     Select  U-Bender
      OUT     B5F0Z1
937   LD      Y5B0Z1
      OR      Y5F0Z1
      OUT     B670Z1
943   LD      SM400  ; Normal  On
      +       K1 Z1
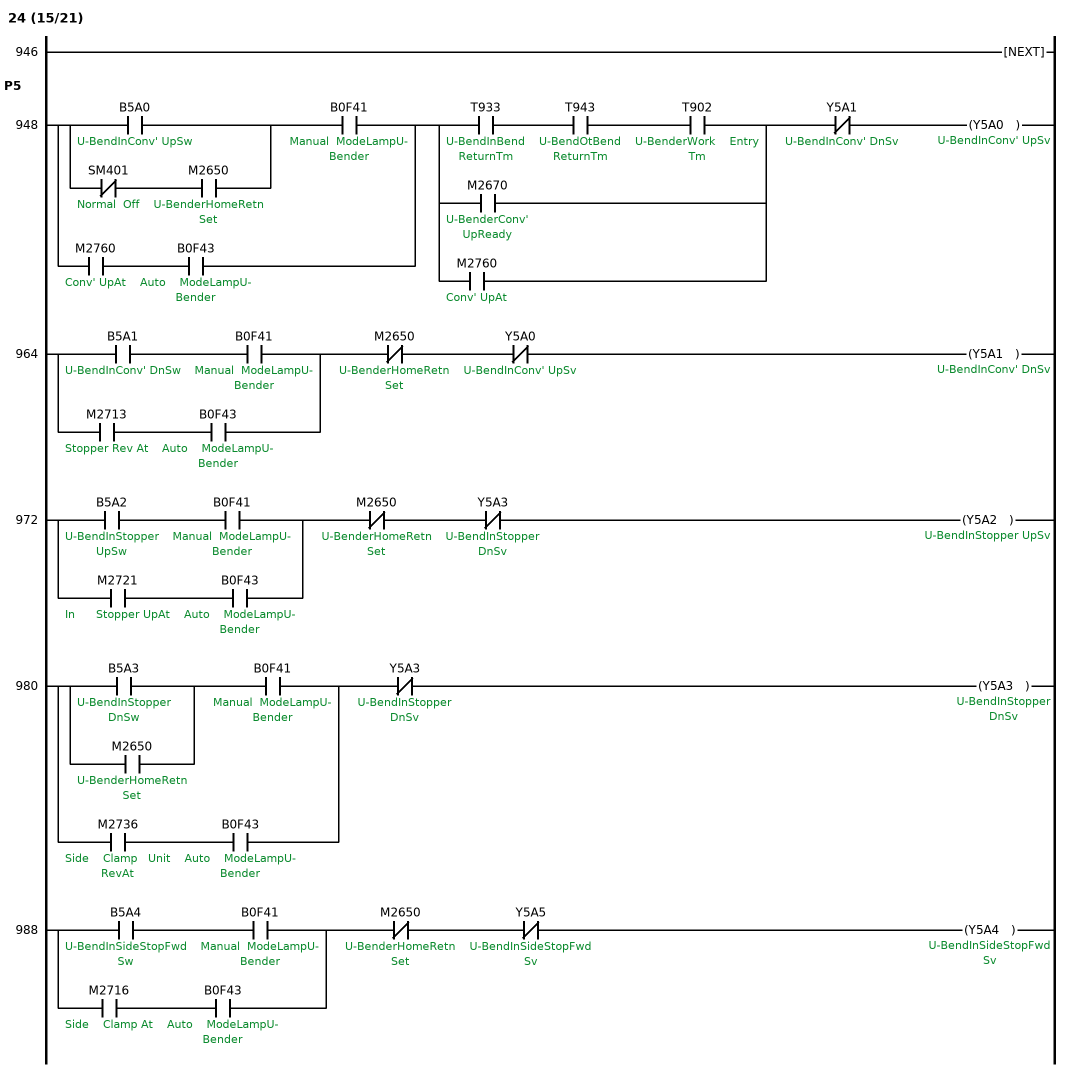
946   NEXT
      P5
948   LD      B5A0  ; U-BendInConv' UpSw
      LDI     SM401  ; Normal  Off
      AND     M2650  ; U-BenderHomeRetnSet
      ORB
      AND     B0F41  ; Manual  ModeLampU-Bender
      LD      M2760  ; Conv' UpAt
      AND     B0F43  ; Auto    ModeLampU-Bender
      ORB
      LD      T933  ; U-BendInBend    ReturnTm
      AND     T943  ; U-BendOtBend    ReturnTm
      AND     T902  ; U-BenderWork    Entry Tm
      OR      M2670  ; U-BenderConv' UpReady
      OR      M2760  ; Conv' UpAt
      ANB
      ANI     Y5A1  ; U-BendInConv' DnSv
      OUT     Y5A0  ; U-BendInConv' UpSv
964   LD      B5A1  ; U-BendInConv' DnSw
      AND     B0F41  ; Manual  ModeLampU-Bender
      LD      M2713  ; Stopper Rev At
      AND     B0F43  ; Auto    ModeLampU-Bender
      ORB
      ANI     M2650  ; U-BenderHomeRetnSet
      ANI     Y5A0  ; U-BendInConv' UpSv
      OUT     Y5A1  ; U-BendInConv' DnSv
972   LD      B5A2  ; U-BendInStopper UpSw
      AND     B0F41  ; Manual  ModeLampU-Bender
      LD      M2721  ; In      Stopper UpAt
      AND     B0F43  ; Auto    ModeLampU-Bender
      ORB
      ANI     M2650  ; U-BenderHomeRetnSet
      ANI     Y5A3  ; U-BendInStopper DnSv
      OUT     Y5A2  ; U-BendInStopper UpSv
980   LD      B5A3  ; U-BendInStopper DnSw
      OR      M2650  ; U-BenderHomeRetnSet
      AND     B0F41  ; Manual  ModeLampU-Bender
      LD      M2736  ; Side    Clamp   Unit RevAt
      AND     B0F43  ; Auto    ModeLampU-Bender
      ORB
      ANI     Y5A3  ; U-BendInStopper DnSv
      OUT     Y5A3  ; U-BendInStopper DnSv
988   LD      B5A4  ; U-BendInSideStopFwd     Sw
      AND     B0F41  ; Manual  ModeLampU-Bender
      LD      M2716  ; Side    Clamp At
      AND     B0F43  ; Auto    ModeLampU-Bender
      ORB
      ANI     M2650  ; U-BenderHomeRetnSet
      ANI     Y5A5  ; U-BendInSideStopFwd     Sv
      OUT     Y5A4  ; U-BendInSideStopFwd     Sv
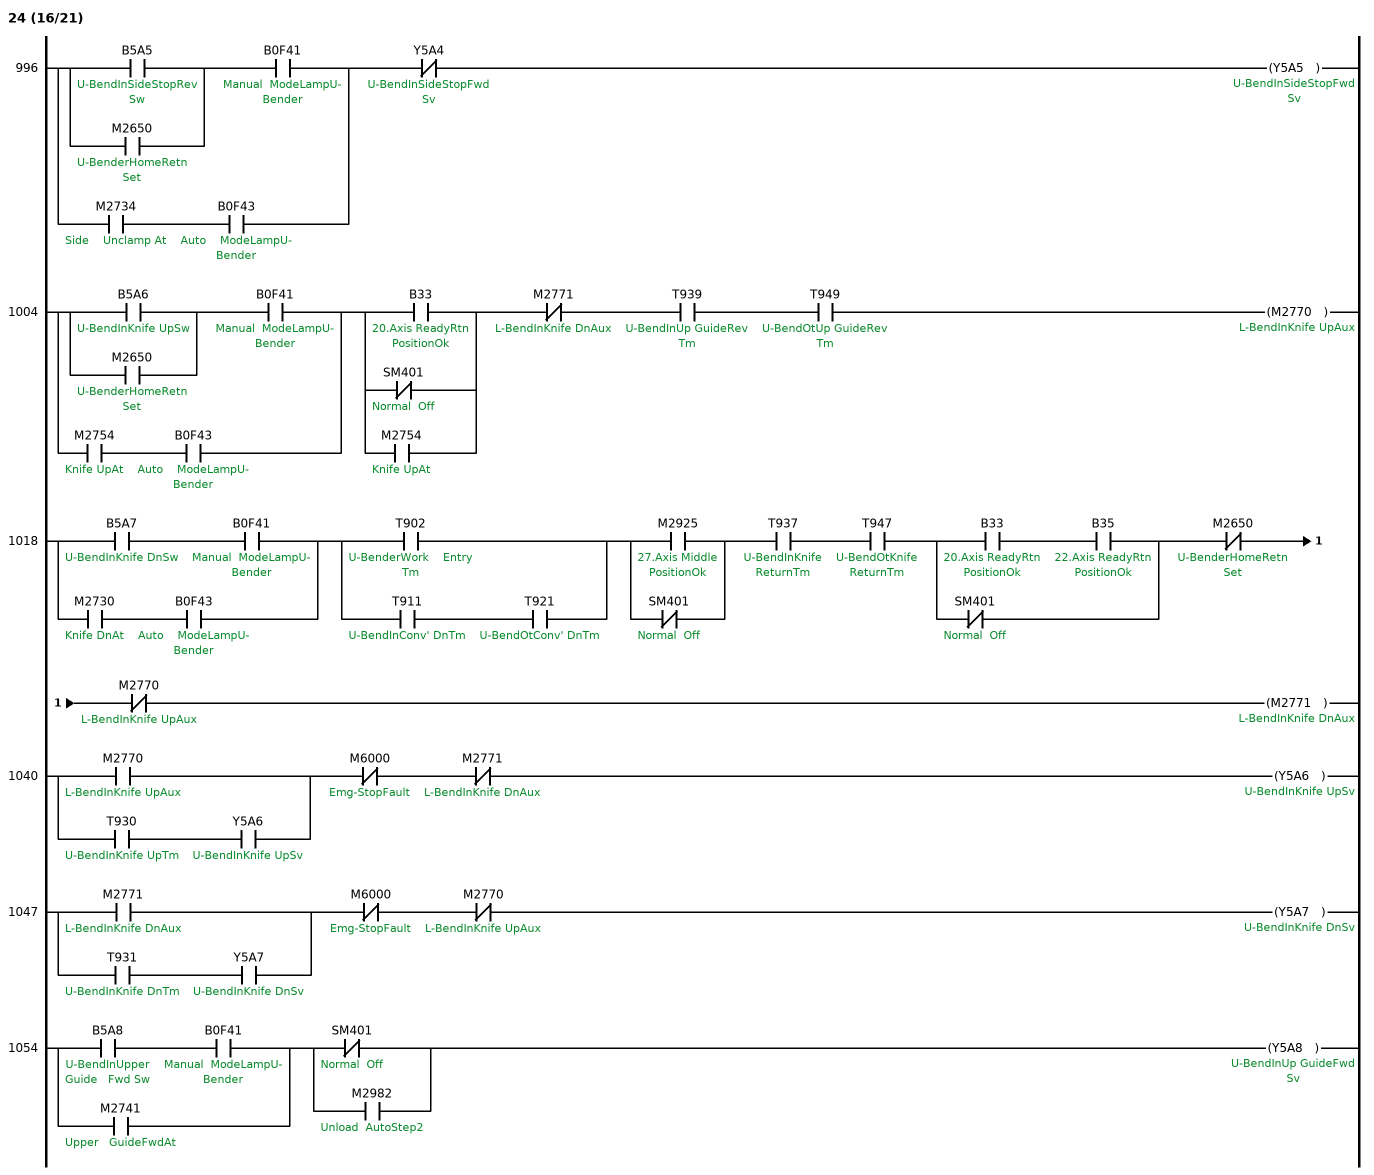
996   LD      B5A5  ; U-BendInSideStopRev     Sw
      OR      M2650  ; U-BenderHomeRetnSet
      AND     B0F41  ; Manual  ModeLampU-Bender
      LD      M2734  ; Side    Unclamp At
      AND     B0F43  ; Auto    ModeLampU-Bender
      ORB
      ANI     Y5A4  ; U-BendInSideStopFwd     Sv
      OUT     Y5A5  ; U-BendInSideStopFwd     Sv
1004  LD      B5A6  ; U-BendInKnife UpSw
      OR      M2650  ; U-BenderHomeRetnSet
      AND     B0F41  ; Manual  ModeLampU-Bender
      LD      M2754  ; Knife UpAt
      AND     B0F43  ; Auto    ModeLampU-Bender
      ORB
      LD      B33  ; 20.Axis ReadyRtnPositionOk
      ORI     SM401  ; Normal  Off
      OR      M2754  ; Knife UpAt
      ANB
      ANI     M2771  ; L-BendInKnife DnAux
      AND     T939  ; U-BendInUp GuideRev Tm
      AND     T949  ; U-BendOtUp GuideRev Tm
      OUT     M2770  ; L-BendInKnife UpAux
1018  LD      B5A7  ; U-BendInKnife DnSw
      AND     B0F41  ; Manual  ModeLampU-Bender
      LD      M2730  ; Knife DnAt
      AND     B0F43  ; Auto    ModeLampU-Bender
      ORB
      LD      T902  ; U-BenderWork    Entry Tm
      LD      T911  ; U-BendInConv' DnTm
      AND     T921  ; U-BendOtConv' DnTm
      ORB
      ANB
      LD      M2925  ; 27.Axis Middle  PositionOk
      ORI     SM401  ; Normal  Off
      ANB
      AND     T937  ; U-BendInKnife   ReturnTm
      AND     T947  ; U-BendOtKnife   ReturnTm
      LD      B33  ; 20.Axis ReadyRtnPositionOk
      AND     B35  ; 22.Axis ReadyRtnPositionOk
      ORI     SM401  ; Normal  Off
      ANB
      ANI     M2650  ; U-BenderHomeRetnSet
      ANI     M2770  ; L-BendInKnife UpAux
      OUT     M2771  ; L-BendInKnife DnAux
1040  LD      M2770  ; L-BendInKnife UpAux
      LD      T930  ; U-BendInKnife UpTm
      AND     Y5A6  ; U-BendInKnife UpSv
      ORB
      ANI     M6000  ; Emg-StopFault
      ANI     M2771  ; L-BendInKnife DnAux
      OUT     Y5A6  ; U-BendInKnife UpSv
1047  LD      M2771  ; L-BendInKnife DnAux
      LD      T931  ; U-BendInKnife DnTm
      AND     Y5A7  ; U-BendInKnife DnSv
      ORB
      ANI     M6000  ; Emg-StopFault
      ANI     M2770  ; L-BendInKnife UpAux
      OUT     Y5A7  ; U-BendInKnife DnSv
1054  LD      B5A8  ; U-BendInUpper   Guide   Fwd Sw
      AND     B0F41  ; Manual  ModeLampU-Bender
      OR      M2741  ; Upper   GuideFwdAt
      LDI     SM401  ; Normal  Off
      OR      M2982  ; Unload  AutoStep2
      ANB
      OUT     Y5A8  ; U-BendInUp GuideFwd Sv
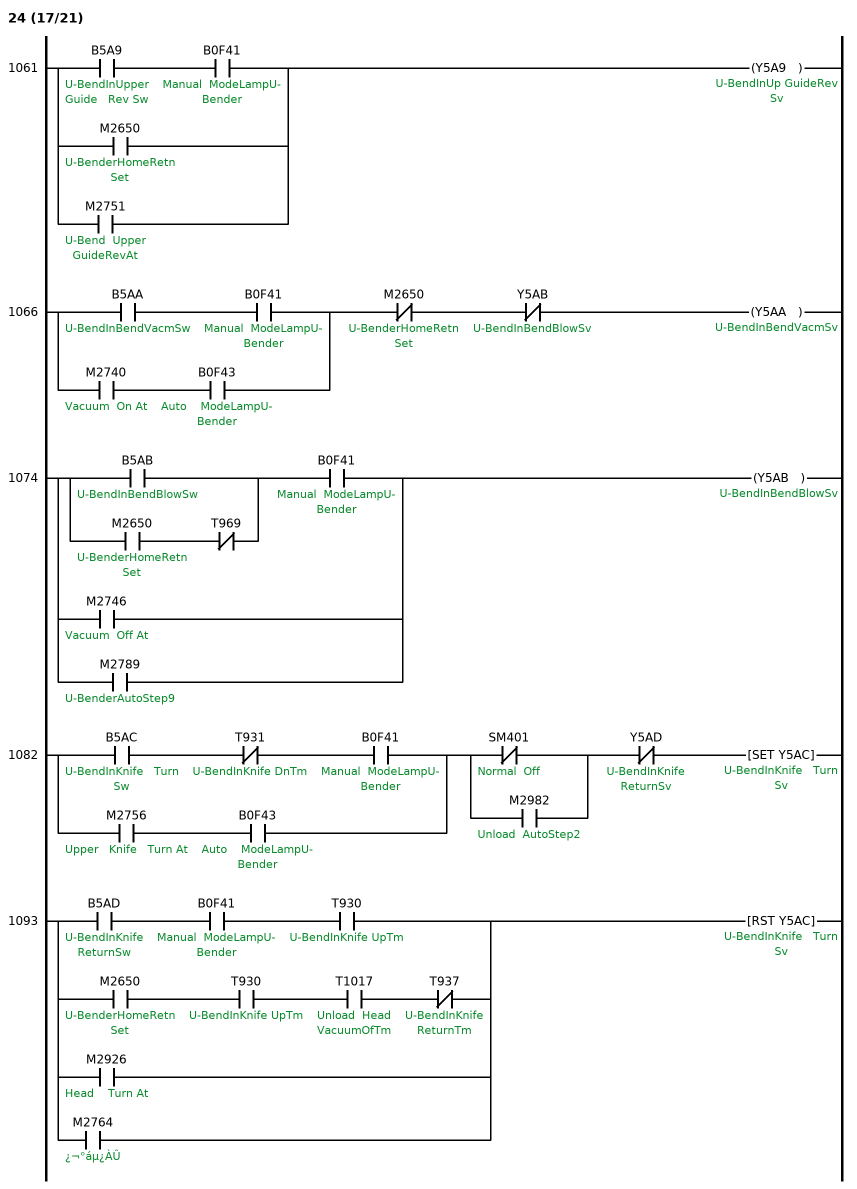
1061  LD      B5A9  ; U-BendInUpper   Guide   Rev Sw
      AND     B0F41  ; Manual  ModeLampU-Bender
      OR      M2650  ; U-BenderHomeRetnSet
      OR      M2751  ; U-Bend  Upper   GuideRevAt
      OUT     Y5A9  ; U-BendInUp GuideRev Sv
1066  LD      B5AA  ; U-BendInBendVacmSw
      AND     B0F41  ; Manual  ModeLampU-Bender
      LD      M2740  ; Vacuum  On At
      AND     B0F43  ; Auto    ModeLampU-Bender
      ORB
      ANI     M2650  ; U-BenderHomeRetnSet
      ANI     Y5AB  ; U-BendInBendBlowSv
      OUT     Y5AA  ; U-BendInBendVacmSv
1074  LD      B5AB  ; U-BendInBendBlowSw
      LD      M2650  ; U-BenderHomeRetnSet
      ANI     T969
      ORB
      AND     B0F41  ; Manual  ModeLampU-Bender
      OR      M2746  ; Vacuum  Off At
      OR      M2789  ; U-BenderAutoStep9
      OUT     Y5AB  ; U-BendInBendBlowSv
1082  LD      B5AC  ; U-BendInKnife   Turn Sw
      ANI     T931  ; U-BendInKnife DnTm
      AND     B0F41  ; Manual  ModeLampU-Bender
      LD      M2756  ; Upper   Knife   Turn At
      AND     B0F43  ; Auto    ModeLampU-Bender
      ORB
      LDI     SM401  ; Normal  Off
      OR      M2982  ; Unload  AutoStep2
      ANB
      ANI     Y5AD  ; U-BendInKnife   ReturnSv
      SET     Y5AC  ; U-BendInKnife   Turn Sv
1093  LD      B5AD  ; U-BendInKnife   ReturnSw
      AND     B0F41  ; Manual  ModeLampU-Bender
      AND     T930  ; U-BendInKnife UpTm
      LD      M2650  ; U-BenderHomeRetnSet
      AND     T930  ; U-BendInKnife UpTm
      AND     T1017  ; Unload  Head    VacuumOfTm
      ANI     T937  ; U-BendInKnife   ReturnTm
      ORB
      OR      M2926  ; Head    Turn At
      OR      M2764  ; ¿¬°áµ¿ÀÛ
      RST     Y5AC  ; U-BendInKnife   Turn Sv
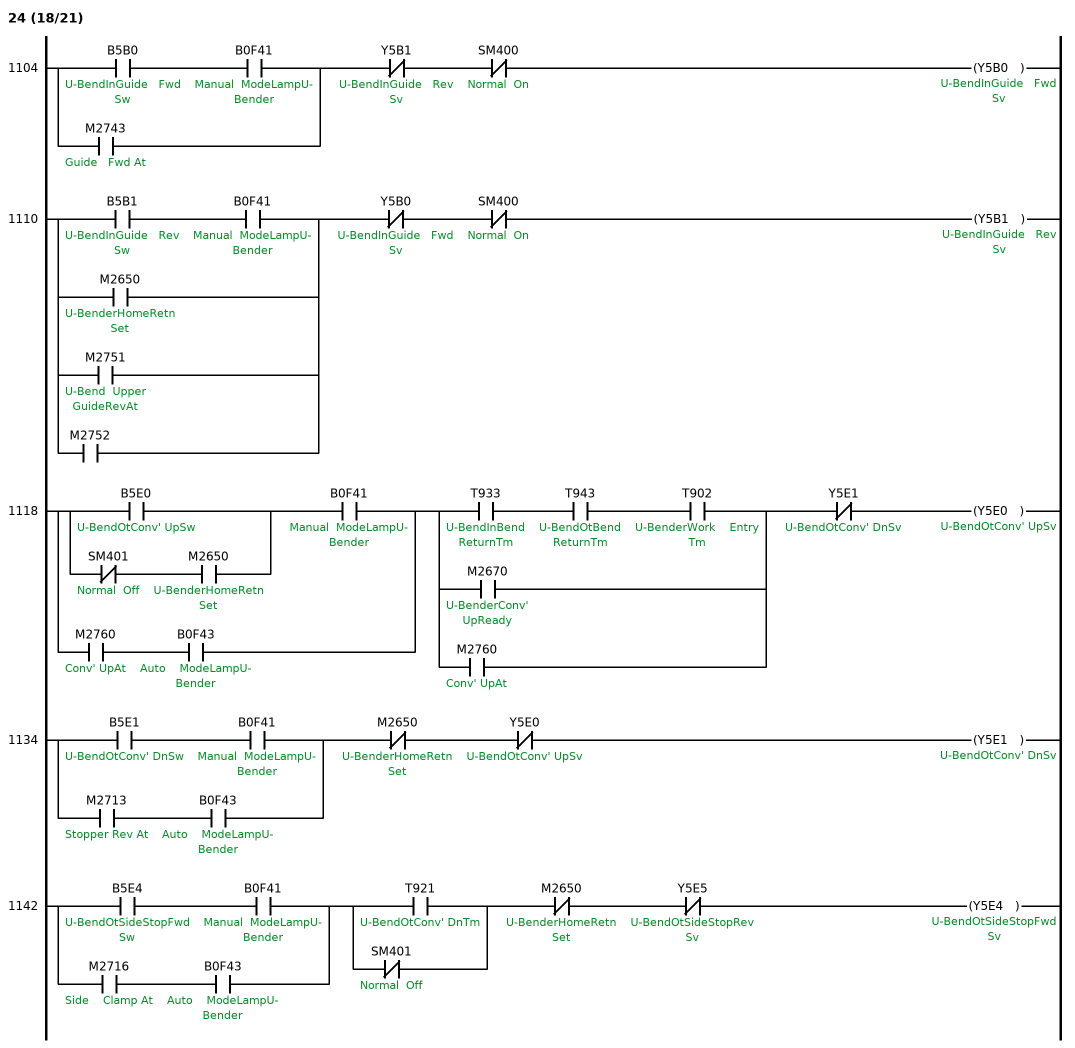
1104  LD      B5B0  ; U-BendInGuide   Fwd Sw
      AND     B0F41  ; Manual  ModeLampU-Bender
      OR      M2743  ; Guide   Fwd At
      ANI     Y5B1  ; U-BendInGuide   Rev Sv
      ANI     SM400  ; Normal  On
      OUT     Y5B0  ; U-BendInGuide   Fwd Sv
1110  LD      B5B1  ; U-BendInGuide   Rev Sw
      AND     B0F41  ; Manual  ModeLampU-Bender
      OR      M2650  ; U-BenderHomeRetnSet
      OR      M2751  ; U-Bend  Upper   GuideRevAt
      OR      M2752
      ANI     Y5B0  ; U-BendInGuide   Fwd Sv
      ANI     SM400  ; Normal  On
      OUT     Y5B1  ; U-BendInGuide   Rev Sv
1118  LD      B5E0  ; U-BendOtConv' UpSw
      LDI     SM401  ; Normal  Off
      AND     M2650  ; U-BenderHomeRetnSet
      ORB
      AND     B0F41  ; Manual  ModeLampU-Bender
      LD      M2760  ; Conv' UpAt
      AND     B0F43  ; Auto    ModeLampU-Bender
      ORB
      LD      T933  ; U-BendInBend    ReturnTm
      AND     T943  ; U-BendOtBend    ReturnTm
      AND     T902  ; U-BenderWork    Entry Tm
      OR      M2670  ; U-BenderConv' UpReady
      OR      M2760  ; Conv' UpAt
      ANB
      ANI     Y5E1  ; U-BendOtConv' DnSv
      OUT     Y5E0  ; U-BendOtConv' UpSv
1134  LD      B5E1  ; U-BendOtConv' DnSw
      AND     B0F41  ; Manual  ModeLampU-Bender
      LD      M2713  ; Stopper Rev At
      AND     B0F43  ; Auto    ModeLampU-Bender
      ORB
      ANI     M2650  ; U-BenderHomeRetnSet
      ANI     Y5E0  ; U-BendOtConv' UpSv
      OUT     Y5E1  ; U-BendOtConv' DnSv
1142  LD      B5E4  ; U-BendOtSideStopFwd     Sw
      AND     B0F41  ; Manual  ModeLampU-Bender
      LD      M2716  ; Side    Clamp At
      AND     B0F43  ; Auto    ModeLampU-Bender
      ORB
      LD      T921  ; U-BendOtConv' DnTm
      ORI     SM401  ; Normal  Off
      ANB
      ANI     M2650  ; U-BenderHomeRetnSet
      ANI     Y5E5  ; U-BendOtSideStopRev     Sv
      OUT     Y5E4  ; U-BendOtSideStopFwd     Sv
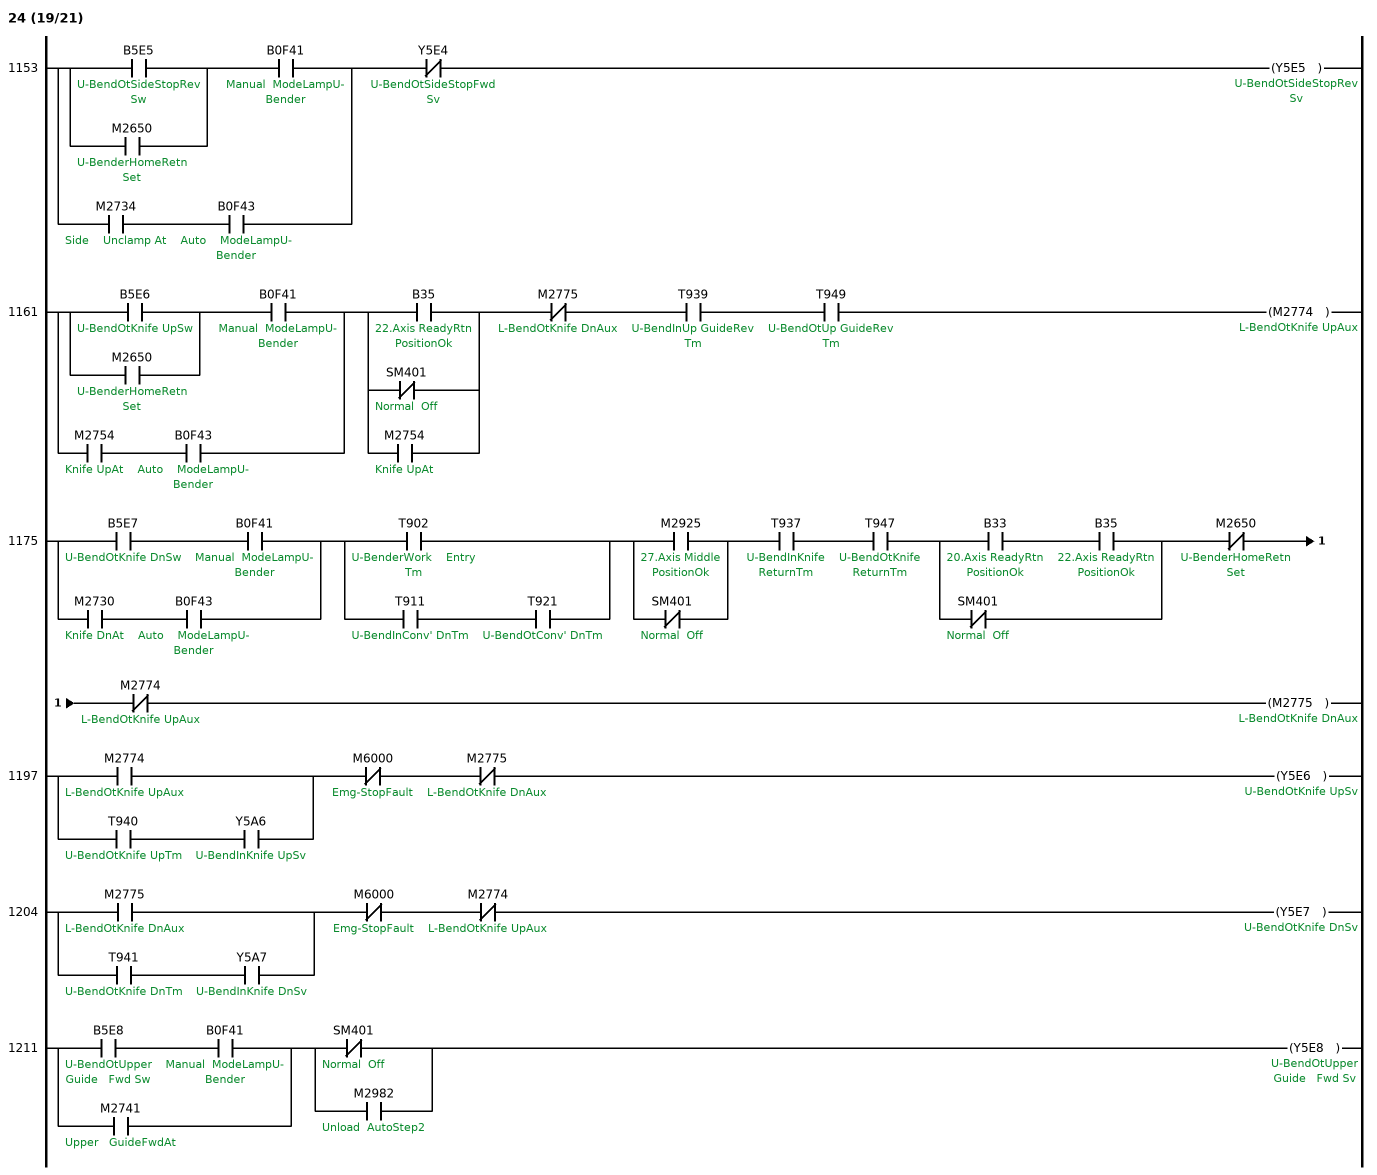
1153  LD      B5E5  ; U-BendOtSideStopRev     Sw
      OR      M2650  ; U-BenderHomeRetnSet
      AND     B0F41  ; Manual  ModeLampU-Bender
      LD      M2734  ; Side    Unclamp At
      AND     B0F43  ; Auto    ModeLampU-Bender
      ORB
      ANI     Y5E4  ; U-BendOtSideStopFwd     Sv
      OUT     Y5E5  ; U-BendOtSideStopRev     Sv
1161  LD      B5E6  ; U-BendOtKnife UpSw
      OR      M2650  ; U-BenderHomeRetnSet
      AND     B0F41  ; Manual  ModeLampU-Bender
      LD      M2754  ; Knife UpAt
      AND     B0F43  ; Auto    ModeLampU-Bender
      ORB
      LD      B35  ; 22.Axis ReadyRtnPositionOk
      ORI     SM401  ; Normal  Off
      OR      M2754  ; Knife UpAt
      ANB
      ANI     M2775  ; L-BendOtKnife DnAux
      AND     T939  ; U-BendInUp GuideRev Tm
      AND     T949  ; U-BendOtUp GuideRev Tm
      OUT     M2774  ; L-BendOtKnife UpAux
1175  LD      B5E7  ; U-BendOtKnife DnSw
      AND     B0F41  ; Manual  ModeLampU-Bender
      LD      M2730  ; Knife DnAt
      AND     B0F43  ; Auto    ModeLampU-Bender
      ORB
      LD      T902  ; U-BenderWork    Entry Tm
      LD      T911  ; U-BendInConv' DnTm
      AND     T921  ; U-BendOtConv' DnTm
      ORB
      ANB
      LD      M2925  ; 27.Axis Middle  PositionOk
      ORI     SM401  ; Normal  Off
      ANB
      AND     T937  ; U-BendInKnife   ReturnTm
      AND     T947  ; U-BendOtKnife   ReturnTm
      LD      B33  ; 20.Axis ReadyRtnPositionOk
      AND     B35  ; 22.Axis ReadyRtnPositionOk
      ORI     SM401  ; Normal  Off
      ANB
      ANI     M2650  ; U-BenderHomeRetnSet
      ANI     M2774  ; L-BendOtKnife UpAux
      OUT     M2775  ; L-BendOtKnife DnAux
1197  LD      M2774  ; L-BendOtKnife UpAux
      LD      T940  ; U-BendOtKnife UpTm
      AND     Y5A6  ; U-BendInKnife UpSv
      ORB
      ANI     M6000  ; Emg-StopFault
      ANI     M2775  ; L-BendOtKnife DnAux
      OUT     Y5E6  ; U-BendOtKnife UpSv
1204  LD      M2775  ; L-BendOtKnife DnAux
      LD      T941  ; U-BendOtKnife DnTm
      AND     Y5A7  ; U-BendInKnife DnSv
      ORB
      ANI     M6000  ; Emg-StopFault
      ANI     M2774  ; L-BendOtKnife UpAux
      OUT     Y5E7  ; U-BendOtKnife DnSv
1211  LD      B5E8  ; U-BendOtUpper   Guide   Fwd Sw
      AND     B0F41  ; Manual  ModeLampU-Bender
      OR      M2741  ; Upper   GuideFwdAt
      LDI     SM401  ; Normal  Off
      OR      M2982  ; Unload  AutoStep2
      ANB
      OUT     Y5E8  ; U-BendOtUpper   Guide   Fwd Sv
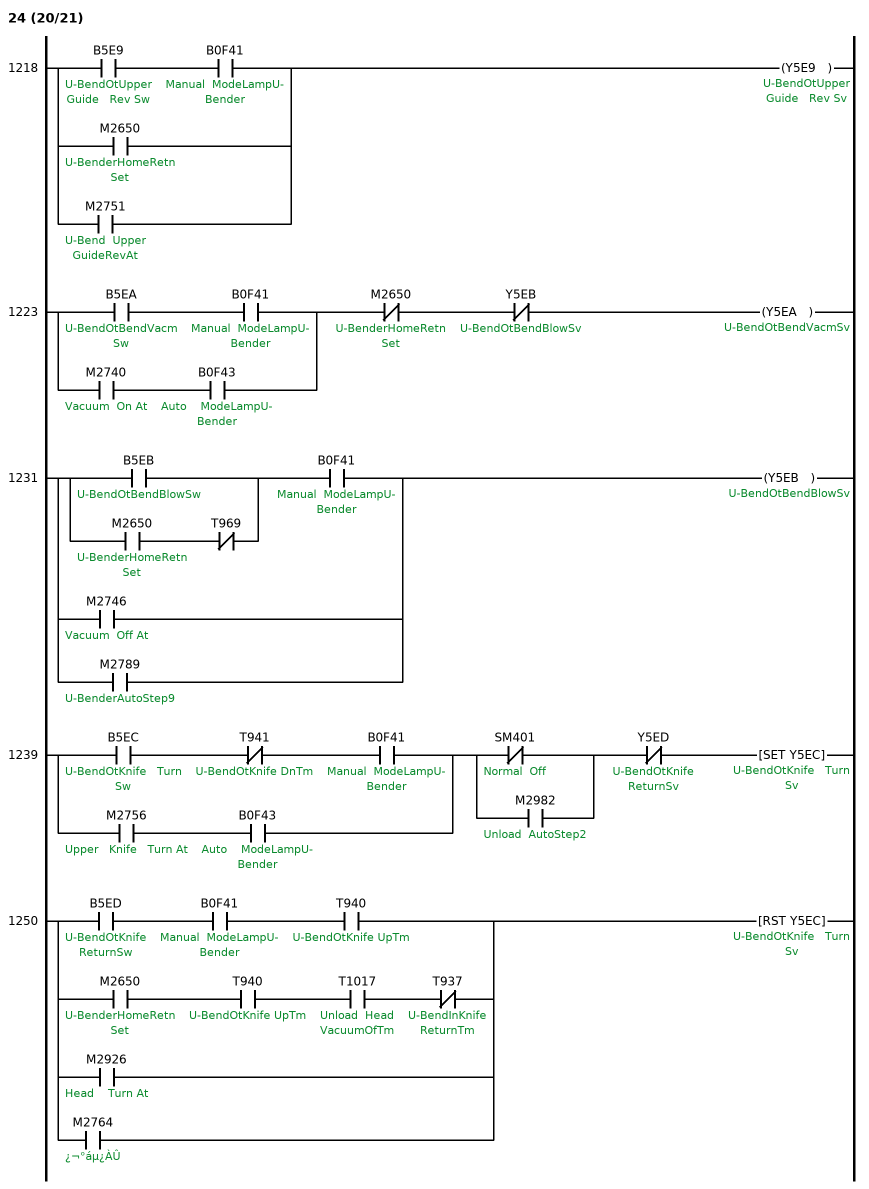
1218  LD      B5E9  ; U-BendOtUpper   Guide   Rev Sw
      AND     B0F41  ; Manual  ModeLampU-Bender
      OR      M2650  ; U-BenderHomeRetnSet
      OR      M2751  ; U-Bend  Upper   GuideRevAt
      OUT     Y5E9  ; U-BendOtUpper   Guide   Rev Sv
1223  LD      B5EA  ; U-BendOtBendVacmSw
      AND     B0F41  ; Manual  ModeLampU-Bender
      LD      M2740  ; Vacuum  On At
      AND     B0F43  ; Auto    ModeLampU-Bender
      ORB
      ANI     M2650  ; U-BenderHomeRetnSet
      ANI     Y5EB  ; U-BendOtBendBlowSv
      OUT     Y5EA  ; U-BendOtBendVacmSv
1231  LD      B5EB  ; U-BendOtBendBlowSw
      LD      M2650  ; U-BenderHomeRetnSet
      ANI     T969
      ORB
      AND     B0F41  ; Manual  ModeLampU-Bender
      OR      M2746  ; Vacuum  Off At
      OR      M2789  ; U-BenderAutoStep9
      OUT     Y5EB  ; U-BendOtBendBlowSv
1239  LD      B5EC  ; U-BendOtKnife   Turn Sw
      ANI     T941  ; U-BendOtKnife DnTm
      AND     B0F41  ; Manual  ModeLampU-Bender
      LD      M2756  ; Upper   Knife   Turn At
      AND     B0F43  ; Auto    ModeLampU-Bender
      ORB
      LDI     SM401  ; Normal  Off
      OR      M2982  ; Unload  AutoStep2
      ANB
      ANI     Y5ED  ; U-BendOtKnife   ReturnSv
      SET     Y5EC  ; U-BendOtKnife   Turn Sv
1250  LD      B5ED  ; U-BendOtKnife   ReturnSw
      AND     B0F41  ; Manual  ModeLampU-Bender
      AND     T940  ; U-BendOtKnife UpTm
      LD      M2650  ; U-BenderHomeRetnSet
      AND     T940  ; U-BendOtKnife UpTm
      AND     T1017  ; Unload  Head    VacuumOfTm
      ANI     T937  ; U-BendInKnife   ReturnTm
      ORB
      OR      M2926  ; Head    Turn At
      OR      M2764  ; ¿¬°áµ¿ÀÛ
      RST     Y5EC  ; U-BendOtKnife   Turn Sv
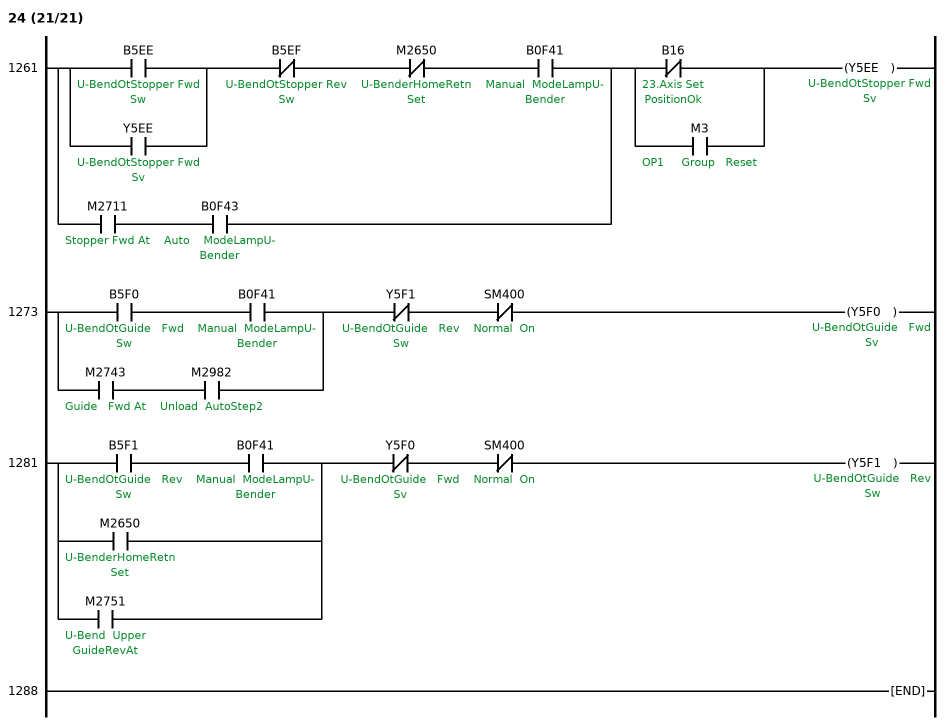
1261  LD      B5EE  ; U-BendOtStopper Fwd Sw
      OR      Y5EE  ; U-BendOtStopper Fwd Sv
      ANI     B5EF  ; U-BendOtStopper Rev Sw
      ANI     M2650  ; U-BenderHomeRetnSet
      AND     B0F41  ; Manual  ModeLampU-Bender
      LD      M2711  ; Stopper Fwd At
      AND     B0F43  ; Auto    ModeLampU-Bender
      ORB
      LDI     B16  ; 23.Axis Set     PositionOk
      OR      M3  ; OP1     Group   Reset
      ANB
      OUT     Y5EE  ; U-BendOtStopper Fwd Sv
1273  LD      B5F0  ; U-BendOtGuide   Fwd Sw
      AND     B0F41  ; Manual  ModeLampU-Bender
      LD      M2743  ; Guide   Fwd At
      AND     M2982  ; Unload  AutoStep2
      ORB
      ANI     Y5F1  ; U-BendOtGuide   Rev Sw
      ANI     SM400  ; Normal  On
      OUT     Y5F0  ; U-BendOtGuide   Fwd Sv
1281  LD      B5F1  ; U-BendOtGuide   Rev Sw
      AND     B0F41  ; Manual  ModeLampU-Bender
      OR      M2650  ; U-BenderHomeRetnSet
      OR      M2751  ; U-Bend  Upper   GuideRevAt
      ANI     Y5F0  ; U-BendOtGuide   Fwd Sv
      ANI     SM400  ; Normal  On
      OUT     Y5F1  ; U-BendOtGuide   Rev Sw
1288  END
END_PROGRAM

PROGRAM 25  // Unload
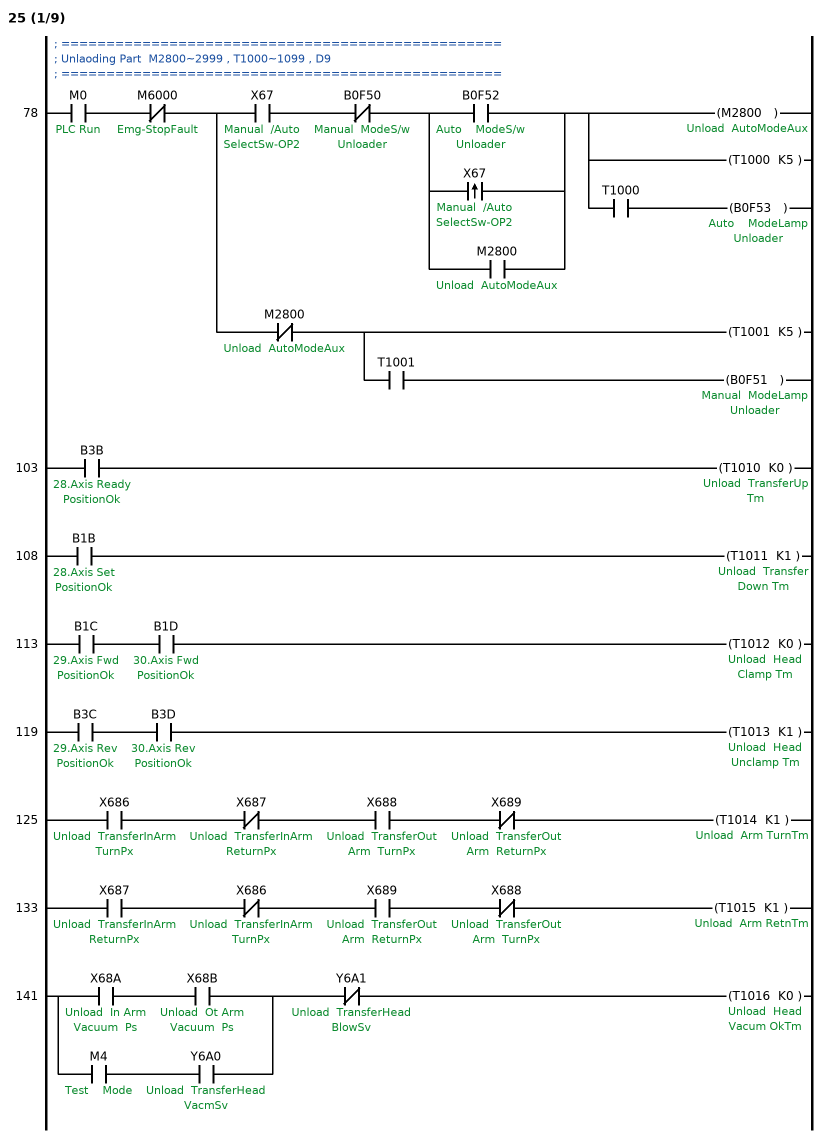
; =================================================
; Unlaoding Part  M2800~2999 , T1000~1099 , D9
; =================================================
78    LD      M0  ; PLC Run
      ANI     M6000  ; Emg-StopFault
      MPS
      AND     X67  ; Manual  /Auto   SelectSw-OP2
      ANI     B0F50  ; Manual  ModeS/w Unloader
      LD      B0F52  ; Auto    ModeS/w Unloader
      ORP     X67  ; Manual  /Auto   SelectSw-OP2
      OR      M2800  ; Unload  AutoModeAux
      ANB
      OUT     M2800  ; Unload  AutoModeAux
      OUT     T1000 K5
      AND     T1000
      OUT     B0F53  ; Auto    ModeLampUnloader
      MPP
      ANI     M2800  ; Unload  AutoModeAux
      OUT     T1001 K5
      AND     T1001
      OUT     B0F51  ; Manual  ModeLampUnloader
103   LD      B3B  ; 28.Axis Ready   PositionOk
      OUT     T1010 K0  ; Unload  TransferUp Tm
108   LD      B1B  ; 28.Axis Set     PositionOk
      OUT     T1011 K1  ; Unload  TransferDown Tm
113   LD      B1C  ; 29.Axis Fwd     PositionOk
      AND     B1D  ; 30.Axis Fwd     PositionOk
      OUT     T1012 K0  ; Unload  Head    Clamp Tm
119   LD      B3C  ; 29.Axis Rev     PositionOk
      AND     B3D  ; 30.Axis Rev     PositionOk
      OUT     T1013 K1  ; Unload  Head    Unclamp Tm
125   LD      X686  ; Unload  TransferInArm   TurnPx
      ANI     X687  ; Unload  TransferInArm   ReturnPx
      AND     X688  ; Unload  TransferOutArm  TurnPx
      ANI     X689  ; Unload  TransferOutArm  ReturnPx
      OUT     T1014 K1  ; Unload  Arm TurnTm
133   LD      X687  ; Unload  TransferInArm   ReturnPx
      ANI     X686  ; Unload  TransferInArm   TurnPx
      AND     X689  ; Unload  TransferOutArm  ReturnPx
      ANI     X688  ; Unload  TransferOutArm  TurnPx
      OUT     T1015 K1  ; Unload  Arm RetnTm
141   LD      X68A  ; Unload  In Arm  Vacuum  Ps
      AND     X68B  ; Unload  Ot Arm  Vacuum  Ps
      LD      M4  ; Test    Mode
      AND     Y6A0  ; Unload  TransferHeadVacmSv
      ORB
      ANI     Y6A1  ; Unload  TransferHeadBlowSv
      OUT     T1016 K0  ; Unload  Head    Vacum OkTm
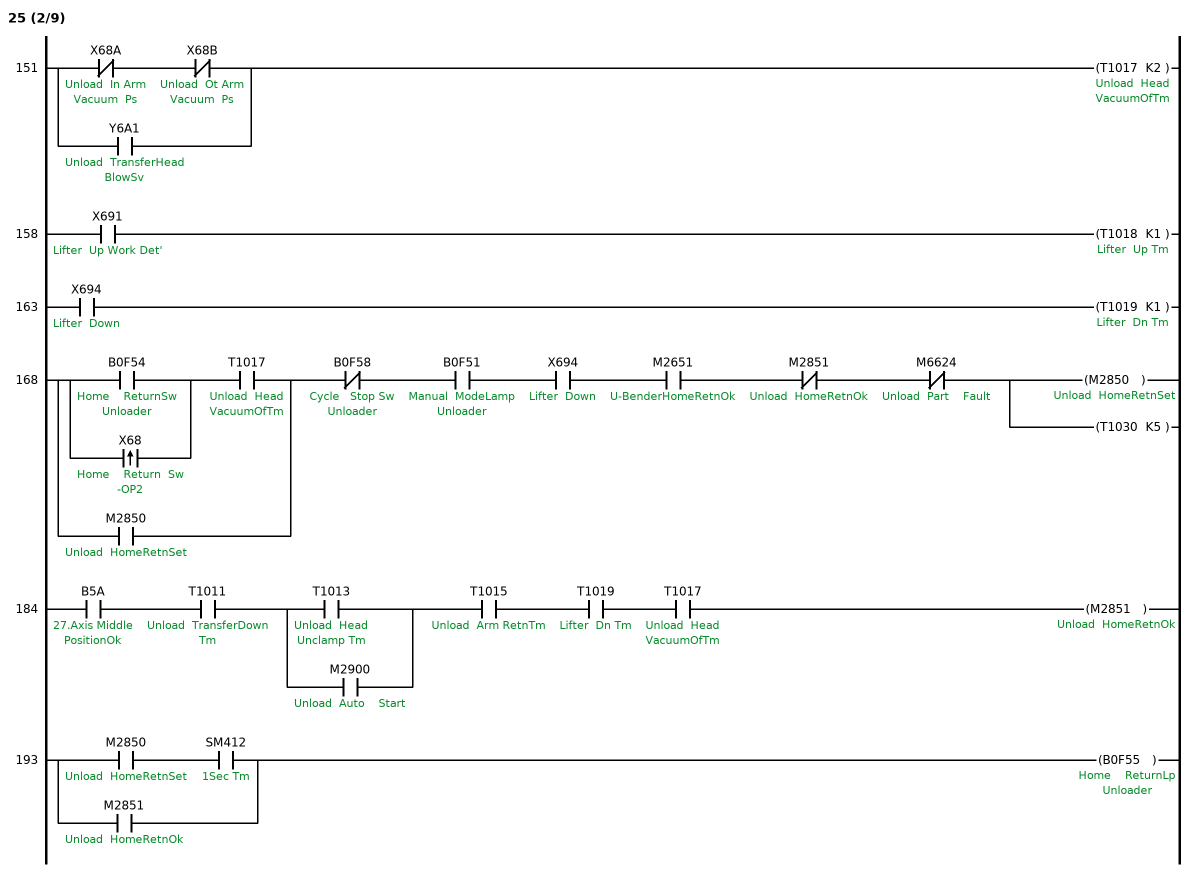
151   LDI     X68A  ; Unload  In Arm  Vacuum  Ps
      ANI     X68B  ; Unload  Ot Arm  Vacuum  Ps
      OR      Y6A1  ; Unload  TransferHeadBlowSv
      OUT     T1017 K2  ; Unload  Head    VacuumOfTm
158   LD      X691  ; Lifter  Up Work Det'
      OUT     T1018 K1  ; Lifter  Up Tm
163   LD      X694  ; Lifter  Down
      OUT     T1019 K1  ; Lifter  Dn Tm
168   LD      B0F54  ; Home    ReturnSwUnloader
      ORP     X68  ; Home    Return  Sw -OP2
      AND     T1017  ; Unload  Head    VacuumOfTm
      OR      M2850  ; Unload  HomeRetnSet
      ANI     B0F58  ; Cycle   Stop Sw Unloader
      AND     B0F51  ; Manual  ModeLampUnloader
      AND     X694  ; Lifter  Down
      AND     M2651  ; U-BenderHomeRetnOk
      ANI     M2851  ; Unload  HomeRetnOk
      ANI     M6624  ; Unload  Part    Fault
      OUT     M2850  ; Unload  HomeRetnSet
      OUT     T1030 K5
184   LD      B5A  ; 27.Axis Middle  PositionOk
      AND     T1011  ; Unload  TransferDown Tm
      LD      T1013  ; Unload  Head    Unclamp Tm
      OR      M2900  ; Unload  Auto    Start
      ANB
      AND     T1015  ; Unload  Arm RetnTm
      AND     T1019  ; Lifter  Dn Tm
      AND     T1017  ; Unload  Head    VacuumOfTm
      OUT     M2851  ; Unload  HomeRetnOk
193   LD      M2850  ; Unload  HomeRetnSet
      AND     SM412  ; 1Sec Tm
      OR      M2851  ; Unload  HomeRetnOk
      OUT     B0F55  ; Home    ReturnLpUnloader
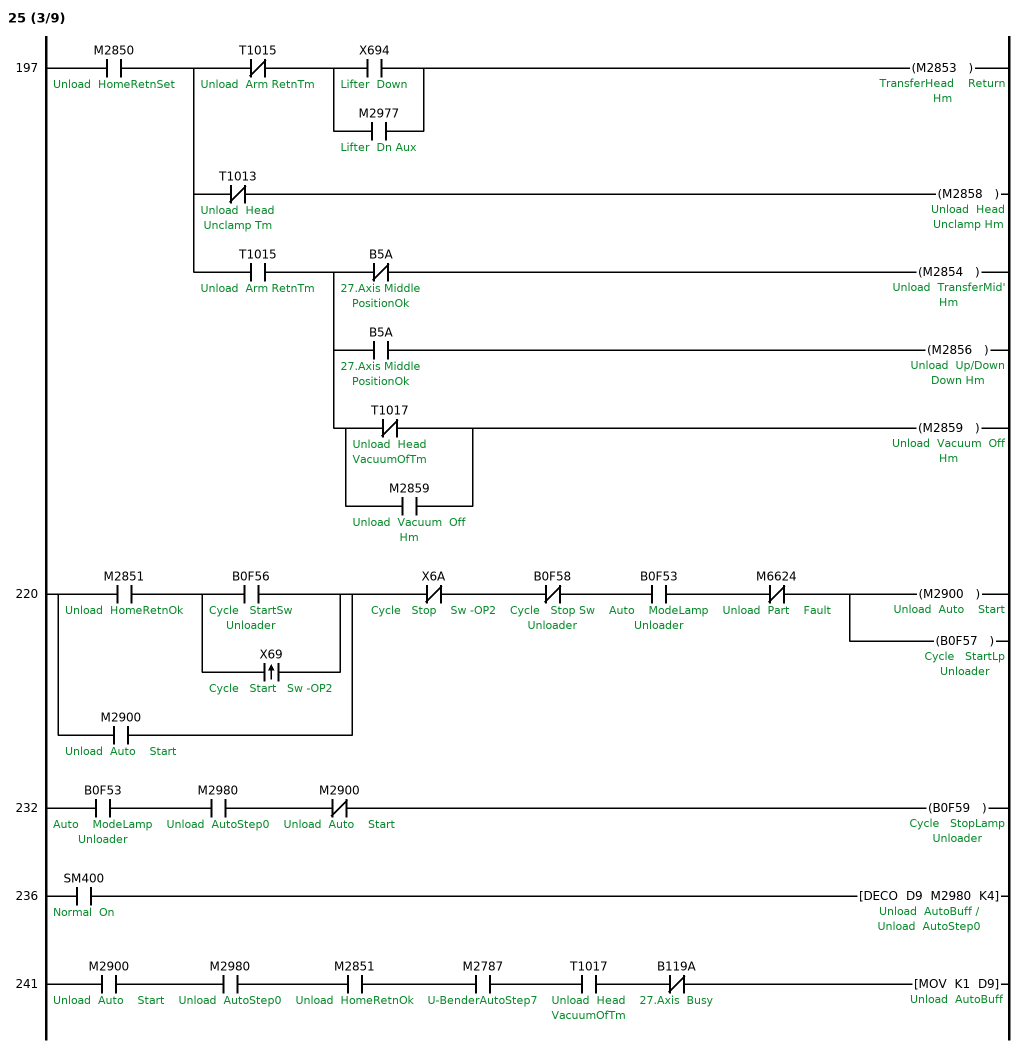
197   LD      M2850  ; Unload  HomeRetnSet
      MPS
      ANI     T1015  ; Unload  Arm RetnTm
      LD      X694  ; Lifter  Down
      OR      M2977  ; Lifter  Dn Aux
      ANB
      OUT     M2853  ; TransferHead    Return  Hm
      MRD
      ANI     T1013  ; Unload  Head    Unclamp Tm
      OUT     M2858  ; Unload  Head    Unclamp Hm
      MPP
      AND     T1015  ; Unload  Arm RetnTm
      MPS
      ANI     B5A  ; 27.Axis Middle  PositionOk
      OUT     M2854  ; Unload  TransferMid' Hm
      MRD
      AND     B5A  ; 27.Axis Middle  PositionOk
      OUT     M2856  ; Unload  Up/Down Down Hm
      MPP
      LDI     T1017  ; Unload  Head    VacuumOfTm
      OR      M2859  ; Unload  Vacuum  Off Hm
      ANB
      OUT     M2859  ; Unload  Vacuum  Off Hm
220   LD      M2851  ; Unload  HomeRetnOk
      LD      B0F56  ; Cycle   StartSw Unloader
      ORP     X69  ; Cycle   Start   Sw -OP2
      ANB
      OR      M2900  ; Unload  Auto    Start
      ANI     X6A  ; Cycle   Stop    Sw -OP2
      ANI     B0F58  ; Cycle   Stop Sw Unloader
      AND     B0F53  ; Auto    ModeLampUnloader
      ANI     M6624  ; Unload  Part    Fault
      OUT     M2900  ; Unload  Auto    Start
      OUT     B0F57  ; Cycle   StartLp Unloader
232   LD      B0F53  ; Auto    ModeLampUnloader
      AND     M2980  ; Unload  AutoStep0
      ANI     M2900  ; Unload  Auto    Start
      OUT     B0F59  ; Cycle   StopLampUnloader
236   LD      SM400  ; Normal  On
      DECO    D9 M2980 K4  ; Unload  AutoBuff
241   LD      M2900  ; Unload  Auto    Start
      AND     M2980  ; Unload  AutoStep0
      AND     M2851  ; Unload  HomeRetnOk
      AND     M2787  ; U-BenderAutoStep7
      AND     T1017  ; Unload  Head    VacuumOfTm
      ANI     B119A  ; 27.Axis  Busy
      MOV     K1 D9
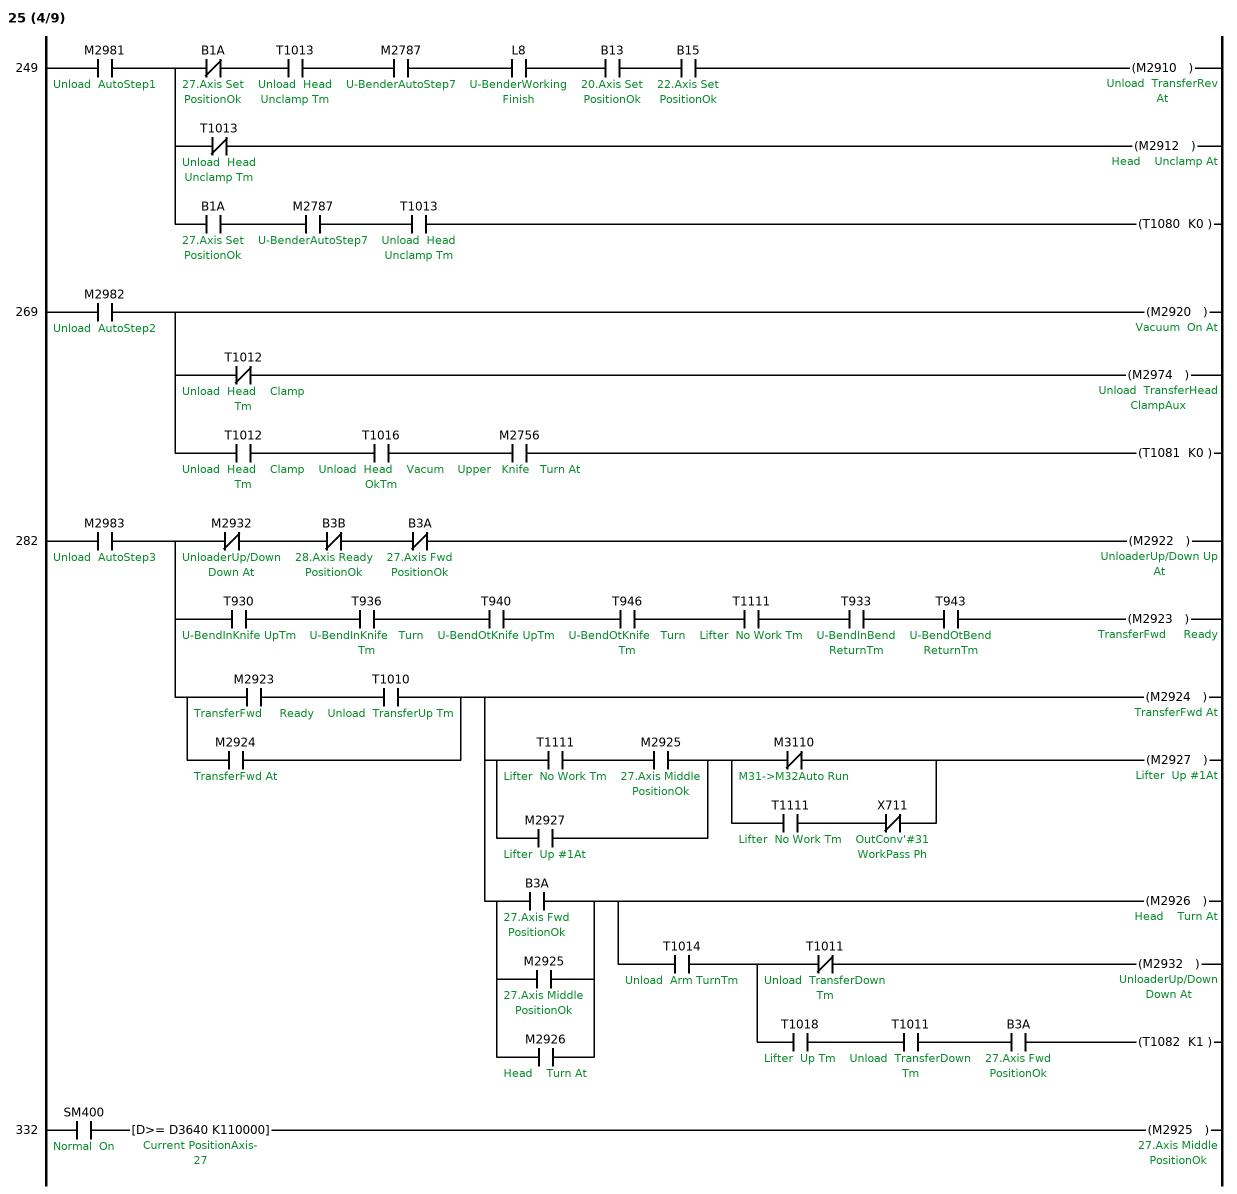
249   LD      M2981  ; Unload  AutoStep1
      MPS
      ANI     B1A  ; 27.Axis Set     PositionOk
      AND     T1013  ; Unload  Head    Unclamp Tm
      AND     M2787  ; U-BenderAutoStep7
      AND     L8  ; U-BenderWorking Finish
      AND     B13  ; 20.Axis Set     PositionOk
      AND     B15  ; 22.Axis Set     PositionOk
      OUT     M2910  ; Unload  TransferRev At
      MRD
      ANI     T1013  ; Unload  Head    Unclamp Tm
      OUT     M2912  ; Head    Unclamp At
      MPP
      AND     B1A  ; 27.Axis Set     PositionOk
      AND     M2787  ; U-BenderAutoStep7
      AND     T1013  ; Unload  Head    Unclamp Tm
      OUT     T1080 K0
269   LD      M2982  ; Unload  AutoStep2
      OUT     M2920  ; Vacuum  On At
      MPS
      ANI     T1012  ; Unload  Head    Clamp Tm
      OUT     M2974  ; Unload  TransferHead    ClampAux
      MPP
      AND     T1012  ; Unload  Head    Clamp Tm
      AND     T1016  ; Unload  Head    Vacum OkTm
      AND     M2756  ; Upper   Knife   Turn At
      OUT     T1081 K0
282   LD      M2983  ; Unload  AutoStep3
      MPS
      ANI     M2932  ; UnloaderUp/Down Down At
      ANI     B3B  ; 28.Axis Ready   PositionOk
      ANI     B3A  ; 27.Axis Fwd     PositionOk
      OUT     M2922  ; UnloaderUp/Down Up At
      MRD
      AND     T930  ; U-BendInKnife UpTm
      AND     T936  ; U-BendInKnife   Turn Tm
      AND     T940  ; U-BendOtKnife UpTm
      AND     T946  ; U-BendOtKnife   Turn Tm
      AND     T1111  ; Lifter  No Work Tm
      AND     T933  ; U-BendInBend    ReturnTm
      AND     T943  ; U-BendOtBend    ReturnTm
      OUT     M2923  ; TransferFwd     Ready
      MPP
      LD      M2923  ; TransferFwd     Ready
      AND     T1010  ; Unload  TransferUp Tm
      OR      M2924  ; TransferFwd At
      ANB
      OUT     M2924  ; TransferFwd At
      MPS
      LD      T1111  ; Lifter  No Work Tm
      AND     M2925  ; 27.Axis Middle  PositionOk
      OR      M2927  ; Lifter  Up #1At
      ANB
      LDI     M3110  ; M31->M32Auto Run
      LD      T1111  ; Lifter  No Work Tm
      ANI     X711  ; OutConv'#31 WorkPass Ph
      ORB
      ANB
      OUT     M2927  ; Lifter  Up #1At
      MPP
      LD      B3A  ; 27.Axis Fwd     PositionOk
      OR      M2925  ; 27.Axis Middle  PositionOk
      OR      M2926  ; Head    Turn At
      ANB
      OUT     M2926  ; Head    Turn At
      AND     T1014  ; Unload  Arm TurnTm
      MPS
      ANI     T1011  ; Unload  TransferDown Tm
      OUT     M2932  ; UnloaderUp/Down Down At
      MPP
      AND     T1018  ; Lifter  Up Tm
      AND     T1011  ; Unload  TransferDown Tm
      AND     B3A  ; 27.Axis Fwd     PositionOk
      OUT     T1082 K1
332   LD      SM400  ; Normal  On
      ANDD>=  D3640 K110000  ; Current PositionAxis-27
      OUT     M2925  ; 27.Axis Middle  PositionOk
